REGION Network 2: Выключение и обнуление таймера
   RUNG wire#powerrail
      I_Contact( #Start )
      wire#w1
      { S7_GenerateENO := "TRUE" } Move(in := 0, out1 => #Now)
      wire#w2
      R_Coil( #"Exit" )
   END_RUNG
   RUNG wire#powerrail
      Contact( #Reset )
   END_RUNG wire#w1
   RUNG wire#powerrail
      { S7_Templates := "SrcType := Int" } LT_Contact(in1 := #Now, in2 := #SP)
   END_RUNG wire#w2
   RUNG wire#w2
      R_Coil( #Reset )
   END_RUNG
   // the same network as SCL:
   // ENO of a box is taken as its EN; it also drops when the box reports an error
   #_w1 := NOT #Start OR #Reset;
   IF #_w1 THEN #Now := 0; END_IF;
   IF #_w1 OR (#Now < #SP) THEN
       #"Exit" := FALSE;
       #Reset := FALSE;
   END_IF;
END_REGION
END_FUNCTION_BLOCK

FUNCTION "Modbus_KP" : Void
{ S7_Optimized_Access := 'TRUE' }
VERSION : 0.1
   VAR_INPUT 
      KP : Int;
      cnt : Int;
   END_VAR

   VAR_OUTPUT 
      use : Bool;
   END_VAR

   VAR_IN_OUT 
      IP {InstructionName := 'IP_V4'; LibVersion := '1.0'} : IP_V4;
      Port : UInt;
      ADDR : UInt;
   END_VAR


BEGIN
	CASE #KP OF
	    1:  //  КП2.1
	        IF NOT "AUMA_KP_2_1_DB".AUMA[#cnt].Use THEN
	            "AUMA_KP_2_1_DB".AUMA[#cnt].Link := FALSE;
	            #use := FALSE;
	        ELSE
	            #use := TRUE;
	            #IP := "tGw_DB".tGw["AUMA_KP_2_1_DB".AUMA[#cnt].ID].IP;
	            #Port := "tGw_DB".tGw["AUMA_KP_2_1_DB".AUMA[#cnt].ID]."Port";
	            #ADDR := "AUMA_KP_2_1_DB".AUMA[#cnt].ADDR;
	        END_IF;
	    2:  //  КП2.2
	        IF NOT "AUMA_KP_2_2_DB".AUMA[#cnt].Use THEN
	            "AUMA_KP_2_2_DB".AUMA[#cnt].Link := FALSE;
	            #use := FALSE;
	        ELSE
	            #use := TRUE;
	            #IP := "tGw_DB".tGw["AUMA_KP_2_2_DB".AUMA[#cnt].ID].IP;
	            #Port := "tGw_DB".tGw["AUMA_KP_2_2_DB".AUMA[#cnt].ID]."Port";
	            #ADDR := "AUMA_KP_2_2_DB".AUMA[#cnt].ADDR;
	        END_IF;
	    3:  //  КП2.3
	        IF NOT "AUMA_KP_2_3_DB".AUMA[#cnt].Use THEN
	            "AUMA_KP_2_3_DB".AUMA[#cnt].Link := FALSE;
	            #use := FALSE;
	        ELSE
	            #use := TRUE;
	            #IP := "tGw_DB".tGw["AUMA_KP_2_3_DB".AUMA[#cnt].ID].IP;
	            #Port := "tGw_DB".tGw["AUMA_KP_2_3_DB".AUMA[#cnt].ID]."Port";
	            #ADDR := "AUMA_KP_2_3_DB".AUMA[#cnt].ADDR;
	        END_IF;
	    4:  //  КП2.4
	        IF NOT "AUMA_KP_2_4_DB".AUMA[#cnt].Use THEN
	            "AUMA_KP_2_4_DB".AUMA[#cnt].Link := FALSE;
	            #use := FALSE;
	        ELSE
	            #use := TRUE;
	            #IP := "tGw_DB".tGw["AUMA_KP_2_4_DB".AUMA[#cnt].ID].IP;
	            #Port := "tGw_DB".tGw["AUMA_KP_2_4_DB".AUMA[#cnt].ID]."Port";
	            #ADDR := "AUMA_KP_2_4_DB".AUMA[#cnt].ADDR;
	        END_IF;
	    5:  //  КП2.5
	        IF NOT "AUMA_KP_2_5_DB".AUMA[#cnt].Use THEN
	            "AUMA_KP_2_5_DB".AUMA[#cnt].Link := FALSE;
	            #use := FALSE;
	        ELSE
	            #use := TRUE;
	            #IP := "tGw_DB".tGw["AUMA_KP_2_5_DB".AUMA[#cnt].ID].IP;
	            #Port := "tGw_DB".tGw["AUMA_KP_2_5_DB".AUMA[#cnt].ID]."Port";
	            #ADDR := "AUMA_KP_2_5_DB".AUMA[#cnt].ADDR;
	        END_IF;
	    6:  //  КП2.6
	        IF NOT "AUMA_KP_2_6_DB".AUMA[#cnt].Use THEN
	            "AUMA_KP_2_6_DB".AUMA[#cnt].Link := FALSE;
	            #use := FALSE;
	        ELSE
	            #use := TRUE;
	            #IP := "tGw_DB".tGw["AUMA_KP_2_6_DB".AUMA[#cnt].ID].IP;
	            #Port := "tGw_DB".tGw["AUMA_KP_2_6_DB".AUMA[#cnt].ID]."Port";
	            #ADDR := "AUMA_KP_2_6_DB".AUMA[#cnt].ADDR;
	        END_IF;
	    7:  //  КП2.7
	        IF NOT "AUMA_KP_2_7_DB".AUMA[#cnt].Use THEN
	            "AUMA_KP_2_7_DB".AUMA[#cnt].Link := FALSE;
	            #use := FALSE;
	        ELSE
	            #use := TRUE;
	            #IP := "tGw_DB".tGw["AUMA_KP_2_7_DB".AUMA[#cnt].ID].IP;
	            #Port := "tGw_DB".tGw["AUMA_KP_2_7_DB".AUMA[#cnt].ID]."Port";
	            #ADDR := "AUMA_KP_2_7_DB".AUMA[#cnt].ADDR;
	        END_IF;
	    8:  //  КП2.8
	        IF NOT "AUMA_KP_2_8_DB".AUMA[#cnt].Use THEN
	            "AUMA_KP_2_8_DB".AUMA[#cnt].Link := FALSE;
	            #use := FALSE;
	        ELSE
	            #use := TRUE;
	            #IP := "tGw_DB".tGw["AUMA_KP_2_8_DB".AUMA[#cnt].ID].IP;
	            #Port := "tGw_DB".tGw["AUMA_KP_2_8_DB".AUMA[#cnt].ID]."Port";
	            #ADDR := "AUMA_KP_2_8_DB".AUMA[#cnt].ADDR;
	        END_IF;
	    9:  //  КП2.9
	        IF NOT "AUMA_KP_2_9_DB".AUMA[#cnt].Use THEN
	            "AUMA_KP_2_9_DB".AUMA[#cnt].Link := FALSE;
	            #use := FALSE;
	        ELSE
	            #use := TRUE;
	            #IP := "tGw_DB".tGw["AUMA_KP_2_9_DB".AUMA[#cnt].ID].IP;
	            #Port := "tGw_DB".tGw["AUMA_KP_2_9_DB".AUMA[#cnt].ID]."Port";
	            #ADDR := "AUMA_KP_2_9_DB".AUMA[#cnt].ADDR;
	        END_IF;
	    10:  //  КП2.10
	        IF NOT "AUMA_KP_2_10_DB".AUMA[#cnt].Use THEN
	            "AUMA_KP_2_10_DB".AUMA[#cnt].Link := FALSE;
	            #use := FALSE;
	        ELSE
	            #use := TRUE;
	            #IP := "tGw_DB".tGw["AUMA_KP_2_10_DB".AUMA[#cnt].ID].IP;
	            #Port := "tGw_DB".tGw["AUMA_KP_2_10_DB".AUMA[#cnt].ID]."Port";
	            #ADDR := "AUMA_KP_2_10_DB".AUMA[#cnt].ADDR;
	        END_IF;
	    11:  //  КП1
	        IF NOT "AUMA_KP_1_DB".AUMA[#cnt].Use THEN
	            "AUMA_KP_1_DB".AUMA[#cnt].Link := FALSE;
	            #use := FALSE;
	        ELSE
	            #use := TRUE;
	            #IP := "tGw_DB".tGw["AUMA_KP_1_DB".AUMA[#cnt].ID].IP;
	            #Port := "tGw_DB".tGw["AUMA_KP_1_DB".AUMA[#cnt].ID]."Port";
	            #ADDR := "AUMA_KP_1_DB".AUMA[#cnt].ADDR;
	        END_IF;
	    ELSE
	        #use := FALSE;
	END_CASE;
END_FUNCTION

FUNCTION "ModBus_AUMA_READ" : Void
{ S7_Optimized_Access := 'TRUE' }
VERSION : 0.1
   VAR_TEMP 
      offset : UInt;
      "DB" : UInt;
   END_VAR


BEGIN
	IF "ModBus_DB".cnt > 0 THEN
	    #offset := ("ModBus_DB".cnt * 40);
	ELSE
	    #offset := 0;
	END_IF;
	
	#DB := 410 + "ModBus_DB".KP;
	
	CASE "ModBus_DB".KP OF
	    1:
	        "AUMA_KP_2_1_DB".AUMA["ModBus_DB".cnt].Link := TRUE;
	        "ModBus_DB".update := "AUMA_KP_2_1_DB".AUMA["ModBus_DB".cnt].Update;
	    2:
	        "AUMA_KP_2_2_DB".AUMA["ModBus_DB".cnt].Link := TRUE;
	        "ModBus_DB".update := "AUMA_KP_2_2_DB".AUMA["ModBus_DB".cnt].Update;
	    3:
	        "AUMA_KP_2_3_DB".AUMA["ModBus_DB".cnt].Link := TRUE;
	        "ModBus_DB".update := "AUMA_KP_2_3_DB".AUMA["ModBus_DB".cnt].Update;
	    4:
	        "AUMA_KP_2_4_DB".AUMA["ModBus_DB".cnt].Link := TRUE;
	        "ModBus_DB".update := "AUMA_KP_2_4_DB".AUMA["ModBus_DB".cnt].Update;
	    5:
	        "AUMA_KP_2_5_DB".AUMA["ModBus_DB".cnt].Link := TRUE;
	        "ModBus_DB".update := "AUMA_KP_2_5_DB".AUMA["ModBus_DB".cnt].Update;
	    6:
	        "AUMA_KP_2_6_DB".AUMA["ModBus_DB".cnt].Link := TRUE;
	        "ModBus_DB".update := "AUMA_KP_2_6_DB".AUMA["ModBus_DB".cnt].Update;
	    7:
	        "AUMA_KP_2_7_DB".AUMA["ModBus_DB".cnt].Link := TRUE;
	        "ModBus_DB".update := "AUMA_KP_2_7_DB".AUMA["ModBus_DB".cnt].Update;
	    8:
	        "AUMA_KP_2_8_DB".AUMA["ModBus_DB".cnt].Link := TRUE;
	        "ModBus_DB".update := "AUMA_KP_2_8_DB".AUMA["ModBus_DB".cnt].Update;
	    9:
	        "AUMA_KP_2_9_DB".AUMA["ModBus_DB".cnt].Link := TRUE;
	        "ModBus_DB".update := "AUMA_KP_2_9_DB".AUMA["ModBus_DB".cnt].Update;
	    10:
	        "AUMA_KP_2_10_DB".AUMA["ModBus_DB".cnt].Link := TRUE;
	        "ModBus_DB".update := "AUMA_KP_2_10_DB".AUMA["ModBus_DB".cnt].Update;
	    11:
	        "AUMA_KP_1_DB".AUMA["ModBus_DB".cnt].Link := TRUE;
	        "ModBus_DB".update := "AUMA_KP_1_DB".AUMA["ModBus_DB".cnt].Update;
	    12:
	        "AUMA_KP_2_DB".AUMA["ModBus_DB".cnt].Link := TRUE;
	        "ModBus_DB".update := "AUMA_KP_2_DB".AUMA["ModBus_DB".cnt].Update;
	    13:
	        "AUMA_KP_3_DB".AUMA["ModBus_DB".cnt].Link := TRUE;
	        "ModBus_DB".update := "AUMA_KP_3_DB".AUMA["ModBus_DB".cnt].Update;
	    14:
	        "AUMA_KP_4_DB".AUMA["ModBus_DB".cnt].Link := TRUE;
	        "ModBus_DB".update := "AUMA_KP_4_DB".AUMA["ModBus_DB".cnt].Update;
	    15:
	        "AUMA_KP_5_DB".AUMA["ModBus_DB".cnt].Link := TRUE;
	        "ModBus_DB".update := "AUMA_KP_5_DB".AUMA["ModBus_DB".cnt].Update;
	END_CASE;
	
	"Indirect_MOVE"(
	                Length := 4,
	                Source_DB := 40,
	                Source_OFFSET := 0,
	                Target_DB := #DB,
	                Target_OFFSET := #offset);
END_FUNCTION

FUNCTION "ModBus_AUMA_ERROR" : Void
{ S7_Optimized_Access := 'TRUE' }
VERSION : 0.1
   VAR_TEMP 
      offset : UInt;
      "DB" : UInt;
   END_VAR


BEGIN
	CASE "ModBus_DB".KP OF
	    1:
	        "AUMA_KP_2_1_DB".AUMA["ModBus_DB".cnt].Link := FALSE;
	        "AUMA_KP_2_1_DB".AUMA["ModBus_DB".cnt].NoRead := TRUE;
	    2:
	        "AUMA_KP_2_2_DB".AUMA["ModBus_DB".cnt].Link := FALSE;
	        "AUMA_KP_2_2_DB".AUMA["ModBus_DB".cnt].NoRead := TRUE;
	    3:
	        "AUMA_KP_2_3_DB".AUMA["ModBus_DB".cnt].Link := FALSE;
	        "AUMA_KP_2_3_DB".AUMA["ModBus_DB".cnt].NoRead := TRUE;
	    4:
	        "AUMA_KP_2_4_DB".AUMA["ModBus_DB".cnt].Link := FALSE;
	        "AUMA_KP_2_4_DB".AUMA["ModBus_DB".cnt].NoRead := TRUE;
	    5:
	        "AUMA_KP_2_5_DB".AUMA["ModBus_DB".cnt].Link := FALSE;
	        "AUMA_KP_2_5_DB".AUMA["ModBus_DB".cnt].NoRead := TRUE;
	    6:
	        "AUMA_KP_2_6_DB".AUMA["ModBus_DB".cnt].Link := FALSE;
	        "AUMA_KP_2_6_DB".AUMA["ModBus_DB".cnt].NoRead := TRUE;
	    7:
	        "AUMA_KP_2_7_DB".AUMA["ModBus_DB".cnt].Link := FALSE;
	        "AUMA_KP_2_7_DB".AUMA["ModBus_DB".cnt].NoRead := TRUE;
	    8:
	        "AUMA_KP_2_8_DB".AUMA["ModBus_DB".cnt].Link := FALSE;
	        "AUMA_KP_2_8_DB".AUMA["ModBus_DB".cnt].NoRead := TRUE;
	    9:
	        "AUMA_KP_2_9_DB".AUMA["ModBus_DB".cnt].Link := FALSE;
	        "AUMA_KP_2_9_DB".AUMA["ModBus_DB".cnt].NoRead := TRUE;
	    10:
	        "AUMA_KP_2_10_DB".AUMA["ModBus_DB".cnt].Link := FALSE;
	        "AUMA_KP_2_10_DB".AUMA["ModBus_DB".cnt].NoRead := TRUE;
	    11:
	        "AUMA_KP_1_DB".AUMA["ModBus_DB".cnt].Link := FALSE;
	        "AUMA_KP_1_DB".AUMA["ModBus_DB".cnt].NoRead := TRUE;
	    12:
	        "AUMA_KP_2_DB".AUMA["ModBus_DB".cnt].Link := FALSE;
	        "AUMA_KP_2_DB".AUMA["ModBus_DB".cnt].NoRead := TRUE;
	    13:
	        "AUMA_KP_3_DB".AUMA["ModBus_DB".cnt].Link := FALSE;
	        "AUMA_KP_3_DB".AUMA["ModBus_DB".cnt].NoRead := TRUE;
	    14:
	        "AUMA_KP_4_DB".AUMA["ModBus_DB".cnt].Link := FALSE;
	        "AUMA_KP_4_DB".AUMA["ModBus_DB".cnt].NoRead := TRUE;
	    15:
	        "AUMA_KP_5_DB".AUMA["ModBus_DB".cnt].Link := FALSE;
	        "AUMA_KP_5_DB".AUMA["ModBus_DB".cnt].NoRead := TRUE;
	    20:
	        "FE_DB".FE["ModBus_DB".cnt].Link := FALSE;
	        "FE_DB".FE["ModBus_DB".cnt].NoRead := TRUE;
	    21:
	        "LE_DB".LE["ModBus_DB".cnt].Link := FALSE;
	        "LE_DB".LE["ModBus_DB".cnt].NoRead := TRUE;
	    22:
	        "PE_DB".PE["ModBus_DB".cnt].Link := FALSE;
	        "PE_DB".PE["ModBus_DB".cnt].NoRead := TRUE;
	END_CASE;
	
	
END_FUNCTION

FUNCTION "ModBus_AUMA_WRITE" : Void
{ S7_Optimized_Access := 'TRUE' }
VERSION : 0.1
   VAR_TEMP 
      offset : UInt;
      "DB" : UInt;
   END_VAR

   VAR CONSTANT 
      I : Byte := 16#81;   // Input
      Q : Byte := 16#82;   // Output
      M : Byte := 16#83;   // Bit Memory
      D : Byte := 16#84;   // Data Block
      PIW : Byte := 16#1;   // S7-1500 Only
      zero : Byte;
   END_VAR


BEGIN
	IF "ModBus_DB".cnt > 0 THEN
	    #offset := ("ModBus_DB".cnt * 40);
	ELSE
	    #offset := 0;
	END_IF;
	
	#DB := 410 + "ModBus_DB".KP;
	
	//запись команды и уставки в коммуникацию
	"Indirect_MOVE"(
	                Length := 2,
	                Source_DB := #DB,
	                Source_OFFSET := #offset + 14,
	                Target_DB := 40,
	                Target_OFFSET := 0);
END_FUNCTION

FUNCTION_BLOCK "ModBus_TCP"   // FB40, LAD
TITLE = Блок опроса ModBus TCP
{ S7_Optimized_Access := 'FALSE' }
VERSION : 0.1
// ВНИМАНИЕ!  Через один аппаратный порт контроллера можно проводить множество различных опросов по ModBus TCP. Для этого у каждого экземпляра должен быть указан уникальный CONNECT.ID.
// 
// Для каждого уникального CONNECT.ID / внешней ветки / точки подключения (IP, RemotePort) рекомендуется использовать отдельный экземпляр функционального блока. Например, при использовании tGW-735 имеющего 3 порта подключения с RemotePort = 502, 503 и 504 соответственно (но общий IP адрес) рекомендуется использовать три отдельных блока ModBus_TCP с уникальными CONNECT.ID.
// 
// Каждая точка чтения/записи = 1 экземпляр DEV_Config, количество элементов в массиве можно менять по необходимости, итоговое количество элементов массива указывается в теге Limit.
// 
// Для режима чтения необходимо указать:
// - MODE = 0
// - Source_DB = 40 (номер DB Modbus_TCP_DB)
// - SourceOFFSET = 0
// - Target_DB = xx (номер DB, куда необходимо положить прочитанные данные)
// - Target_OFFSET = xx (номер байта, начиная с которого кладутся прочитанные данные в выбранный DB)
// 
// Для режима опроса необходимо указать:
// - MODE = 1
// - Source_DB = xx (номер DB, откуда необходимо взять данные для передачи)
// - Source_OFFSET = xx (номер байта, начиная с которого берутся данные для передачи)
// - Target_DB = 40 (номер DB Modbus_TCP_DB)
// - Target_OFFSET = 0
// stored: AutoNumber false, IsIECCheckEnabled false, SetENOAutomatically false, UDAEnableTagReadback false
   VAR DB_SPECIFIC
      DATA : Array[0..100] of Word;   // Массив данных
      CONNECT { S7_SetPoint := 'True'} : TCON_IP_v4;
   END_VAR
   // CONNECT.InterfaceId := 64;
   // CONNECT.ID := 16#0001;
   // CONNECT.ConnectionType := 16#0B;
   // CONNECT.ActiveEstablished := TRUE;
   // CONNECT.RemoteAddress.ADDR[1] := 16#C0;
   // CONNECT.RemoteAddress.ADDR[2] := 16#A8;
   // CONNECT.RemoteAddress.ADDR[3] := 16#00;
   // CONNECT.RemoteAddress.ADDR[4] := 16#0A;
   // CONNECT.RemotePort := 502;
   // CONNECT.LocalPort := 0;
BEGIN

REGION Network 1
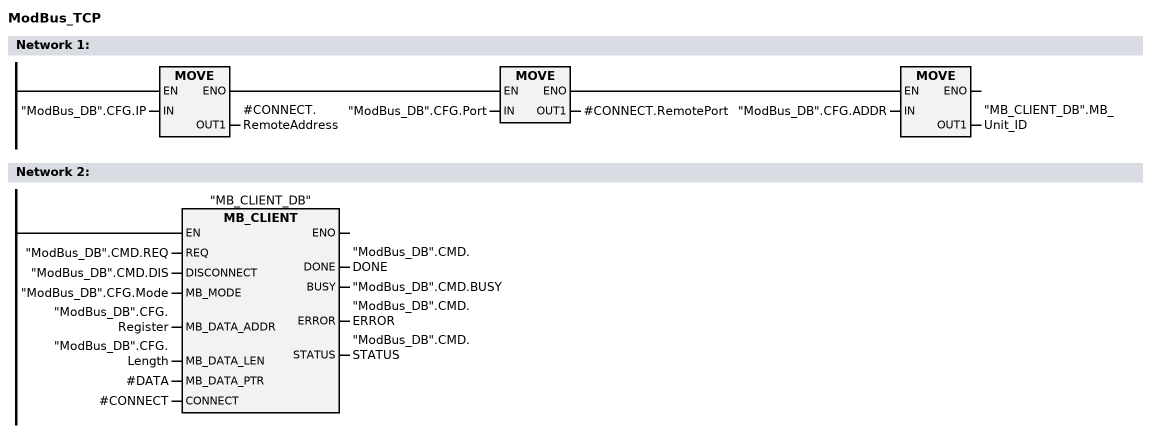
   RUNG wire#powerrail
      Move(in := "ModBus_DB".CFG.IP, out1 => #CONNECT.RemoteAddress)
      Move(in := "ModBus_DB".CFG.Port, out1 => #CONNECT.RemotePort)
      Move(in := "ModBus_DB".CFG.ADDR, out1 => "MB_CLIENT_DB".MB_Unit_ID)
   END_RUNG
   // the same network as SCL:
   #CONNECT.RemoteAddress := "ModBus_DB".CFG.IP;
   #CONNECT.RemotePort := "ModBus_DB".CFG.Port;
   "MB_CLIENT_DB".MB_Unit_ID := "ModBus_DB".CFG.ADDR;
END_REGION

REGION Network 2
   RUNG wire#powerrail
      "MB_CLIENT_DB".MB_CLIENT(REQ := "ModBus_DB".CMD.REQ, DISCONNECT := "ModBus_DB".CMD.DIS, MB_MODE := "ModBus_DB".CFG.Mode, MB_DATA_ADDR := "ModBus_DB".CFG.Register, MB_DATA_LEN := "ModBus_DB".CFG.Length, MB_DATA_PTR := #DATA, CONNECT := #CONNECT, DONE => "ModBus_DB".CMD.DONE, BUSY => "ModBus_DB".CMD.BUSY, ERROR => "ModBus_DB".CMD.ERROR, STATUS => "ModBus_DB".CMD.STATUS)
   END_RUNG
   // the same network as SCL:
   "MB_CLIENT_DB"(REQ := "ModBus_DB".CMD.REQ,   // MB_CLIENT
                  DISCONNECT := "ModBus_DB".CMD.DIS,
                  MB_MODE := "ModBus_DB".CFG.Mode,
                  MB_DATA_ADDR := "ModBus_DB".CFG.Register,
                  MB_DATA_LEN := "ModBus_DB".CFG.Length,
                  MB_DATA_PTR := #DATA,
                  CONNECT := #CONNECT,
                  DONE => "ModBus_DB".CMD.DONE,
                  BUSY => "ModBus_DB".CMD.BUSY,
                  ERROR => "ModBus_DB".CMD.ERROR,
                  STATUS => "ModBus_DB".CMD.STATUS);
END_REGION
END_FUNCTION_BLOCK

FUNCTION_BLOCK "SKV_Main"
{ S7_Optimized_Access := 'FALSE' }
VERSION : 0.1
   VAR 
      One : Array[0..11] of "SKV_One";
      SP : Struct   // Уставки
         Max { S7_SetPoint := 'True'} : Real;   // - максимальная производительность
         High : Real;   // - высокая производительность
         Auto : Real;   // - рабочая уставка
         Point : Real;   // - сниженная производительность
         Low : Real;   // - низкая производительность
         Min { S7_SetPoint := 'True'} : Real;   // - минимальная производительность
      END_STRUCT;
      cnt : Struct   // счетчики
         Min { S7_SetPoint := 'True'} : Int;   // - минимальное кол-во устр-в
         Fix { S7_SetPoint := 'True'} : Int := 2;   // - кол-во устр-в в фиксированном режиме
         All : Int;   // - кол-во устройств общее
         Group : Int;   // - кол-во основных устройств
         Reserve : Int;   // - кол-во резервных устройств
         Ready : Int;   // - кол-во готовых устройств
         Low : Int;   // - кол-во устр-в на сниженной скорости
         Work : Int;   // - кол-во запущенных устройств
         Start : Int;   // - кол-во устр-в в работе
      END_STRUCT;
      tmp : Int;
   END_VAR


BEGIN
	//Распредление нагрузки
	"SKV_Load"(Add_REQ :="SKV_cnt_DB".CMD.Add,
	           Add_Ready => "SKV_cnt_DB".Data.Add_Ready,
	           cnt := #tmp);
	
	//Управление запуском и остановом
	"SKV_cnt_DB"();
	
	//Выбор кол-ва устр-в
	"SKV_Logic_DB"();
	
	//Проверка готовности маршрутов
	"Route_Check_DB"();
	
	//управление маршрутами
	"Route_Control_DB"();
	
	REGION "SKV_One"
	    // Вызов управления каждой скважиной
	    #One[1](Ready:= "Comm_SKV_1".From_SKV.STATE.Ready,
	            Warning:= "Comm_SKV_1".From_SKV.STATE.Warning,
	            Alarm:= "Comm_SKV_1".From_SKV.STATE.Alarm,
	            Route:="Comm_SKV_1".Route,
	            FeedBack := "Comm_SKV_1".FE,
	            REQ_CMD=> "Comm_SKV_1".To_SKV.CMD.REQ,
	            REQ_SP=> "Comm_SKV_1".SP_FE);
	    #One[2](Ready := "Comm_SKV_2".From_SKV.STATE.Ready,
	            Warning := "Comm_SKV_2".From_SKV.STATE.Warning,
	            Alarm := "Comm_SKV_2".From_SKV.STATE.Alarm,
	            Route := "Comm_SKV_2".Route,
	            FeedBack := "Comm_SKV_2".FE,
	            REQ_CMD => "Comm_SKV_2".To_SKV.CMD.REQ,
	            REQ_SP => "Comm_SKV_2".SP_FE);
	    #One[3](Ready := "Comm_SKV_3".From_SKV.STATE.Ready,
	            Warning := "Comm_SKV_3".From_SKV.STATE.Warning,
	            Alarm := "Comm_SKV_3".From_SKV.STATE.Alarm,
	            Route := "Comm_SKV_3".Route,
	            FeedBack := "Comm_SKV_3".FE,
	            REQ_CMD => "Comm_SKV_3".To_SKV.CMD.REQ,
	            REQ_SP => "Comm_SKV_3".SP_FE);
	    #One[4](Ready := "Comm_SKV_12".From_SKV.STATE.Ready,
	            Warning := "Comm_SKV_12".From_SKV.STATE.Warning,
	            Alarm := "Comm_SKV_12".From_SKV.STATE.Alarm,
	            Route := "Comm_SKV_12".Route,
	            FeedBack := "Comm_SKV_12".FE,
	            REQ_CMD => "Comm_SKV_12".To_SKV.CMD.REQ,
	            REQ_SP => "Comm_SKV_12".SP_FE);
	    #One[5](Ready := "Comm_SKV_13".From_SKV.STATE.Ready,
	            Warning := "Comm_SKV_13".From_SKV.STATE.Warning,
	            Alarm := "Comm_SKV_13".From_SKV.STATE.Alarm,
	            Route := "Comm_SKV_13".Route,
	            FeedBack := "Comm_SKV_13".FE,
	            REQ_CMD => "Comm_SKV_13".To_SKV.CMD.REQ,
	            REQ_SP => "Comm_SKV_13".SP_FE);
	    #One[6](Ready := "Comm_SKV_14".From_SKV.STATE.Ready,
	            Warning := "Comm_SKV_14".From_SKV.STATE.Warning,
	            Alarm := "Comm_SKV_14".From_SKV.STATE.Alarm,
	            Route := "Comm_SKV_14".Route,
	            FeedBack := "Comm_SKV_14".FE,
	            REQ_CMD => "Comm_SKV_14".To_SKV.CMD.REQ,
	            REQ_SP => "Comm_SKV_14".SP_FE);
	    #One[7](Ready := "Comm_SKV_15".From_SKV.STATE.Ready,
	            Warning := "Comm_SKV_15".From_SKV.STATE.Warning,
	            Alarm := "Comm_SKV_15".From_SKV.STATE.Alarm,
	            Route := "Comm_SKV_15".Route,
	            FeedBack := "Comm_SKV_15".FE,
	            REQ_CMD => "Comm_SKV_15".To_SKV.CMD.REQ,
	            REQ_SP => "Comm_SKV_15".SP_FE);
	    #One[8](Ready := "Comm_SKV_20".From_SKV.STATE.Ready,
	            Warning := "Comm_SKV_20".From_SKV.STATE.Warning,
	            Alarm := "Comm_SKV_20".From_SKV.STATE.Alarm,
	            Route := "Comm_SKV_20".Route,
	            FeedBack := "Comm_SKV_20".FE,
	            REQ_CMD => "Comm_SKV_20".To_SKV.CMD.REQ,
	            REQ_SP => "Comm_SKV_20".SP_FE);
	    #One[9](Ready := "Comm_SKV_21".From_SKV.STATE.Ready,
	            Warning := "Comm_SKV_21".From_SKV.STATE.Warning,
	            Alarm := "Comm_SKV_21".From_SKV.STATE.Alarm,
	            Route := "Comm_SKV_21".Route,
	            FeedBack := "Comm_SKV_21".FE,
	            REQ_CMD => "Comm_SKV_21".To_SKV.CMD.REQ,
	            REQ_SP => "Comm_SKV_21".SP_FE);
	    #One[10](Ready := "Comm_SKV_22".From_SKV.STATE.Ready,
	             Warning := "Comm_SKV_22".From_SKV.STATE.Warning,
	             Alarm := "Comm_SKV_22".From_SKV.STATE.Alarm,
	             Route := "Comm_SKV_22".Route,
	             FeedBack := "Comm_SKV_22".FE,
	             REQ_CMD => "Comm_SKV_22".To_SKV.CMD.REQ,
	             REQ_SP => "Comm_SKV_22".SP_FE);
	    #One[11](Ready := "Comm_SKV_23".From_SKV.STATE.Ready,
	             Warning := "Comm_SKV_23".From_SKV.STATE.Warning,
	             Alarm := "Comm_SKV_23".From_SKV.STATE.Alarm,
	             Route := "Comm_SKV_23".Route,
	             FeedBack := "Comm_SKV_23".FE,
	             REQ_CMD => "Comm_SKV_23".To_SKV.CMD.REQ,
	             REQ_SP => "Comm_SKV_23".SP_FE);
	END_REGION
	
END_FUNCTION_BLOCK

FUNCTION_BLOCK "SKV_One"
{ S7_Optimized_Access := 'FALSE' }
VERSION : 0.1
   VAR_INPUT 
      Ready : Bool;   // Флаг готовности устр-ва
      Warning : Bool;   // Флаг предупрждения
      Alarm : Bool;   // Флаг аварии устр-ва
      Route : Bool;   // Флаг готовности маршрута
      FeedBack : Real;   // ОС производительности утр-ва
   END_VAR

   VAR_OUTPUT 
      REQ_CMD : Bool;   // Команда - запуск устр-ва
      REQ_SP : Real;   // Команда - уставка производительности устр-ва
   END_VAR

   VAR 
      Enable : Bool;   // Флаг выбора устр-ва для работы
      SP_Use { S7_SetPoint := 'True'} : Bool := true;   // Использовать флаг достижения уставки
      CMD { S7_SetPoint := 'False'} : "CMD";   // Управляющее слово
      Mode { S7_SetPoint := 'True'} : Int;   // Режим работы
      Status : Int;   // Статус устр-ва
      C { S7_SetPoint := 'True'} : Real;   // Коэффециент эффективности
      Delta : Real;   // Текущее отклонение от уставки
      SP : Struct   // Уставки
         Ok : Bool;   // Флаг достижения уставки
         Auto : Real;   // - авто режим
         Hand : Real;   // - ручной режим
         Low_Percent { S7_SetPoint := 'True'} : Real := 85.0;   // - замедление до %
         Low : Real;   // - замедленная скорость
         Min { S7_SetPoint := 'True'} : Real := 30.0;   // - минимальный расход
         Max { S7_SetPoint := 'True'} : Real := 45.0;   // - максимальный расход
         Delta { S7_SetPoint := 'True'} : Real := 10.0;   // - допустимое отклонение
         Last : Real;   // - прошлая уставка
      END_STRUCT;
      drv_CMD { S7_SetPoint := 'False'} : "drv_CMD";
      support : Word;
      PT {InstructionName := 'R_TRIG'; LibVersion := '1.0'; S7_SetPoint := 'False'} : Array[0..1] of R_TRIG;
      NT {InstructionName := 'F_TRIG'; LibVersion := '1.0'; S7_SetPoint := 'False'} : Array[0..1] of F_TRIG;
   END_VAR


BEGIN
	//Управление одной скважиной
	
	#CMD.Lock := NOT #Ready OR #Alarm;  //Запрет запуска
	#CMD.Ready := NOT #CMD.Lock;
	
	//Ограничение уставки
	IF NOT #CMD.Hand THEN
	    #SP.Hand := #SP.Auto;
	END_IF;
	IF #SP.Hand < #SP.Min THEN
	    #SP.Hand := #SP.Min;
	END_IF;
	IF #SP.Hand > #SP.Max THEN
	    #SP.Hand := #SP.Max;
	END_IF;
	
	//Замедленная скорость
	#SP.Low := #SP.Hand * (100 / #SP.Low_Percent);
	
	//Контроль достижения уставки
	IF #SP.Last <> #SP.Hand THEN
	    #Delta := ABS(#SP.Hand - #SP.Last);
	    IF #Delta < #SP.Delta THEN
	        #SP.Last := #SP.Hand;
	        #SP.Ok := TRUE;
	    ELSE
	        #SP.Ok := FALSE;
	    END_IF;
	END_IF;
	#PT[0](CLK := #SP.Ok);
	
	//device control
	#drv_CMD(Emergency := #support.%X0,
	          CMD := #CMD);
	 //manual mode flag
	     IF #CMD.Hand THEN
	         "Hand_MDA" := TRUE;
	     END_IF;
	     
	//Отключение
	     IF NOT #CMD.Start_M AND #Mode > 1 AND #Mode <= 5 THEN
	         IF #Status <> 5 THEN
	             #Mode := 5;
	         ELSE
	             #Mode := 6;
	         END_IF;
	     END_IF;
	     
	//Режимы работы
	     CASE #Mode OF
	         0: //Установка отключена
	             #CMD.Start_A := FALSE;
	             #CMD.Start_M := FALSE;
	             #Status := 0;
	             #Mode := 1;
	         1: //Запуск в работу
	             IF #CMD.Start_M THEN
	                 #REQ_CMD := TRUE;
	                 #REQ_SP := #SP.Min;
	                 IF #Status = 0 THEN
	                     #Status := 10; //выход на минимальную рабочую точку
	                 ELSIF #Status = 10 AND (#PT[0].Q OR NOT #SP_Use) THEN
	                     #Status := 1;  //готов к работе
	                 END_IF;
	             ELSE
	                 #REQ_CMD := FALSE;
	                 #REQ_SP := 0.0;
	                 #Status := 0;
	             END_IF;
	         2:  //Плавный разгон до общей точки
	             IF #Status = 1 THEN
	                 #REQ_SP := #SP.Hand;
	                 #Status := 20;     //выход на общую рабочую точку
	             ELSIF #Status = 20 AND (#PT[0].Q OR NOT #SP_Use) THEN
	                 #Status := 2;      //рабочая точка достигнута
	             END_IF;
	         3:  //Переход в штатный режим работы
	             IF #Status = 2 OR #Status = 4 THEN
	                 #Status := 3;       //штатный режим работы
	             ELSIF #Status = 3 THEN
	                 IF NOT #Warning THEN
	                     #REQ_SP := #SP.Hand;
	                 ELSE
	                     #REQ_SP := #SP.Low;
	                 END_IF;
	             END_IF;
	         4: //Замедление перед вводном нового элемента в работу
	             IF #Status = 3 THEN
	                 #REQ_SP := #SP.Hand;
	                 #Status := 40;        //замедление при вводе нового элемента
	             ELSIF #Status = 40 AND (#PT[0].Q OR NOT #SP_Use) THEN
	                 #Status := 4;
	             END_IF;
	         5: //Замедление при отключении
	             IF #Status <> 50 AND #Status <> 5 THEN
	                 #REQ_SP := #SP.Min;
	                 #Status := 50;
	             ELSIF #Status = 50 AND (NOT #Enable OR #CMD.Lock OR (#PT[0].Q OR NOT #SP_Use)) THEN
	                 #Status := 5;
	             END_IF;
	         6: //Вывод элемента из работы
	             IF #Status = 5 THEN
	                 #CMD.Start_A := FALSE;
	                 #REQ_CMD := FALSE;
	                 #REQ_SP := 0.0;
	                 #Status := 60;
	             ELSIF #Status = 60 AND (#PT[0].Q OR NOT #SP_Use) THEN
	                 #Status := 0;
	                 #Mode := 0;
	             END_IF;
	     END_CASE;
	     
	
END_FUNCTION_BLOCK

FUNCTION_BLOCK "drv_CMD"
{ S7_Optimized_Access := 'TRUE' }
VERSION : 0.1
   VAR_INPUT 
      Emergency : Bool;
   END_VAR

   VAR_IN_OUT 
      CMD : "CMD";
   END_VAR


BEGIN
	// Device mode determination
	IF NOT #Emergency THEN
	    //Normal mode
	    IF NOT #CMD.Force THEN
	        //No technological lock
	        IF NOT #CMD.Lock AND NOT #CMD.Alarm THEN
	            //No manual mode
	            IF NOT #CMD.Hand THEN
	                #CMD.Start_M := #CMD.Start_A;
	            END_IF;
	        ELSE
	            //Technological lock or device alarm
	            #CMD.Start_M := FALSE;
	        END_IF;
	    ELSE
	        IF #CMD.Lock OR #CMD.Alarm THEN
	            #CMD.Start_M := FALSE;
	        END_IF;
	    END_IF;
	ELSE
	    //Emergency stop
	    #CMD.Start_M := FALSE;
	END_IF;
END_FUNCTION_BLOCK

FUNCTION "SKV_Load" : Void
{ S7_Optimized_Access := 'TRUE' }
VERSION : 0.1
   VAR_INPUT 
      Add_REQ : Bool;   // Запрос ввода нового устр-ва в работу
   END_VAR

   VAR_OUTPUT 
      Add_Ready : Bool;   // Устр-ва готовы к вводу нового устр-ва в работу
   END_VAR

   VAR_IN_OUT 
      cnt : Int;   // счетчик
   END_VAR

   VAR_TEMP 
      x : Int;
   END_VAR


BEGIN
	//обнуление временных значений
	#Add_Ready := FALSE;
	"SKV_Main_DB".cnt.Ready := 0;
	"SKV_Main_DB".cnt.Low := 0;
	"SKV_Main_DB".cnt.Start := 0;
	"SKV_Main_DB".cnt.Work := 0;
	
	IF "SKV_Main_DB".SP.Auto > "SKV_Main_DB".SP.Max THEN
	    "SKV_Main_DB".SP.Auto := "SKV_Main_DB".SP.Max;
	END_IF;
	
	//вычисление точки схождения скоростей
	"SKV_Main_DB".SP.Point := "SKV_Main_DB".SP.Low + ((("SKV_Main_DB".SP.Auto - "SKV_Main_DB".SP.Low) / "SKV_Main_DB".cnt.Min) * 2);
	
	//Распределение уставки по работающим насосам
	FOR #x := 1 TO "SKV_Main_DB".cnt.All DO
	    
	    //число готовых насосов
	    IF "SKV_Main_DB".One[#x].CMD.Ready THEN
	        "SKV_Main_DB".cnt.Ready := "SKV_Main_DB".cnt.Ready + 1;
	    END_IF;
	    
	    //число насосов в работе
	    IF "SKV_Main_DB".One[#x].CMD.Start_M THEN
	        "SKV_Main_DB".cnt.Start := "SKV_Main_DB".cnt.Start + 1;
	    END_IF;
	    
	    //число насосов в штатном режиме
	    IF "SKV_Main_DB".One[#x].Status = 3 THEN
	        "SKV_Main_DB".cnt.Work := "SKV_Main_DB".cnt.Work + 1;
	    END_IF;
	    
	    //запуск установки
	    IF "SKV_cnt_DB".Step > 0 THEN
	        IF "SKV_cnt_DB".Step < 10 THEN
	            IF "SKV_Main_DB".One[#x].Status = 1 THEN
	                "SKV_Main_DB".One[#x].Mode := 2;
	            END_IF;
	            IF "SKV_Main_DB".One[#x].Status = 2 THEN
	                "SKV_Main_DB".One[#x].Mode := 3;
	            END_IF;
	            "SKV_Main_DB".One[#x].SP.Auto := "SKV_Main_DB".SP.Auto;
	        END_IF;
	    END_IF;
	    
	    //уставка в рабочем режиме
	    IF "SKV_Main_DB".One[#x].Status = 3 OR "SKV_Main_DB".One[#x].Status = 30 THEN
	        "SKV_Main_DB".One[#x].SP.Auto := "SKV_Main_DB".SP.Auto;
	    END_IF;
	    
	  //цикл замедления при подключении нового насоса
	    IF #Add_REQ THEN
	        
	        //команда замедлиться для подключения работающих насосов
	        IF "SKV_Main_DB".One[#x].Status = 3 THEN
	            "SKV_Main_DB".One[#x].Mode := 4;
	        END_IF;
	        
	        //коррекция уставки для замедленных насосов
	        IF "SKV_Main_DB".One[#x].Status = 40 THEN
	            "SKV_Main_DB".One[#x].SP.Auto := "SKV_Main_DB".SP.Point;
	        END_IF;
	        
	        //контроль готовности всех насосов
	        IF "SKV_Main_DB".One[#x].Status = 4 THEN
	            "SKV_Main_DB".cnt.Low := "SKV_Main_DB".cnt.Low + 1;
	            IF "SKV_Main_DB".cnt.Low = #cnt THEN
	                #Add_Ready := true;
	            END_IF;
	        END_IF;
	        
	    END_IF;
	    
	    //возвращение в рабочий режим
	    IF NOT #Add_REQ THEN
	        IF "SKV_Main_DB".One[#x].Status = 4 THEN
	            "SKV_Main_DB".One[#x].Mode := 3;
	        END_IF;
	    END_IF;
	    
	END_FOR;
	
END_FUNCTION

FUNCTION_BLOCK "SKV_Logic"
{ S7_Optimized_Access := 'FALSE' }
VERSION : 0.1
   VAR 
      Start : Bool;   // Команда запуска
      Start_Up { S7_SetPoint := 'True'} : Bool;   // Авто-рестарт
      Mode : Bool;   // Режим работы
      Step : Int;   // шаг операции
      LE : Real;   // Текущий усреднённый уровень
      SP : Struct   // Уставки
         Max { S7_SetPoint := 'True'} : Real;   // - макс уровень
         High { S7_SetPoint := 'True'} : Real;   // - высокий уровень
         Mid { S7_SetPoint := 'True'} : Real;   // - средний уровень
         Low { S7_SetPoint := 'True'} : Real;   // - низкий уровень
         Min { S7_SetPoint := 'True'} : Real;   // - минимальный уровень
      END_STRUCT;
   END_VAR


BEGIN
	//Отключение при первом пуске
	IF NOT #Start_Up AND "FirstScan" THEN
	    #Start := FALSE;
	END_IF;
	
	//Отключение
	IF NOT #Start THEN
	    #Step := 0;
	    "SKV_cnt_DB".CMD.REQ := 0;
	END_IF;
	
	//Общее управление
	CASE #Step OF
	    0:  //Запуск системы
	        IF #Start AND #LE < #SP.Max THEN
	            "SKV_cnt_DB".CMD.REQ := "SKV_Main_DB".cnt.Min;  //минимальное количество устр-в в работе
	            #Step := #Step + 1;
	        END_IF;
	    1:  //проверка режима
	        IF #Mode = 0 THEN
	            #Step := 2; //поддержание уровня
	        ELSIF #Mode = 1 THEN
	            #Step := 3; //фиксированная нагрузка
	        END_IF;
	    2:  //Поддержание уровня
	        IF #LE < #SP.High THEN                              //уровень ниже верхней рабочей точки - вошли в рабочий диапазон
	            IF #LE < #SP.Mid THEN                           //уровень упал ниже среднего - требуется +1 устр-во
	                IF "SKV_cnt_DB".CMD.REQ = "SKV_Main_DB".cnt.Work THEN
	                    IF "SKV_Main_DB".cnt.Work < "SKV_Main_DB".cnt.All AND "SKV_cnt_DB".Step = 10 THEN
	                        "SKV_cnt_DB".CMD.REQ := "SKV_cnt_DB".CMD.REQ + 1;
	                    END_IF;
	                END_IF;
	                IF NOT "SKV_cnt_DB".CMD.Reload AND NOT NOT "SKV_cnt_DB".CMD.Load AND NOT "SKV_cnt_DB".CMD.Rotation AND NOT "SKV_cnt_DB".CMD.Deload AND "SKV_cnt_DB".Step = 10 THEN
	                    IF "SKV_cnt_DB".CMD.REQ > "SKV_Main_DB".cnt.Start THEN
	                        "SKV_cnt_DB".CMD.Reload := TRUE;
	                    END_IF;
	                    IF "SKV_cnt_DB".CMD.REQ < "SKV_Main_DB".cnt.Start THEN
	                        "SKV_cnt_DB".CMD.Deload := TRUE;
	                    END_IF;
	                END_IF;
	            END_IF;
	        ELSE
	            IF "SKV_cnt_DB".CMD.REQ = "SKV_Main_DB".cnt.Work AND "SKV_cnt_DB".Step = 10 THEN
	                "SKV_cnt_DB".CMD.REQ := "SKV_cnt_DB".CMD.REQ - 1;
	                (*IF "SKV_cnt_DB".CMD.REQ < "SKV_Main_DB".cnt.Min THEN
	                    "SKV_cnt_DB".CMD.REQ := "SKV_Main_DB".cnt.Min;
	                END_IF;*)
	                IF "SKV_cnt_DB".CMD.REQ < 0 THEN
	                    "SKV_cnt_DB".CMD.REQ := 0;
	                END_IF;
	            END_IF;
	        END_IF;
	        //Смена режима работы
	        IF #Mode <> 0 THEN
	            #Step := 1;
	        END_IF;
	    3:   //Фиксированный режим
	        IF NOT "SKV_cnt_DB".CMD.Reload AND NOT NOT "SKV_cnt_DB".CMD.Load AND NOT "SKV_cnt_DB".CMD.Rotation AND NOT "SKV_cnt_DB".CMD.Deload AND "SKV_cnt_DB".Step = 10 THEN
	            IF "SKV_cnt_DB".CMD.REQ > "SKV_Main_DB".cnt.Start THEN
	                "SKV_cnt_DB".CMD.Reload := TRUE;
	            END_IF;
	            IF "SKV_cnt_DB".CMD.REQ < "SKV_Main_DB".cnt.Start THEN
	                "SKV_cnt_DB".CMD.Deload := TRUE;
	            END_IF;
	        END_IF;
	        //Смена режима работы
	        IF #Mode <> 1 THEN
	            #Step := 1;
	        END_IF;
	END_CASE;
END_FUNCTION_BLOCK

FUNCTION_BLOCK "KP_2_1"
{ S7_Optimized_Access := 'FALSE' }
VERSION : 0.1
   VAR 
      limit { S7_SetPoint := 'True'} : Int := 2;   // число задвижек в камере
      load : Int;   // отображаемые на экране настройки
      load_last : Int;
      KP : Array[0..10] of "DRV_AUMA";
      load_ok { S7_SetPoint := 'True'} : Bool;
   END_VAR

   VAR_TEMP 
      ID : Int;
      cnt : Int;
   END_VAR


BEGIN
	//дистанционный режим управления
	FOR #cnt := 1 TO #limit BY 1 DO
	    IF "Comm_SKV_2".To_SKV.Valves.Local[0] THEN
	        IF #KP[#cnt].CMD.Hand THEN
	            #KP[#cnt].CMD.Start_M := "Comm_SKV_2".From_SKV.Valves.REQ[#cnt];
	        END_IF;
	        IF "Comm_SKV_2".From_SKV.Valves.REQ[0] THEN
	            #KP[#cnt].CMD.Reset := TRUE;
	            #load := 10;
	        END_IF;
	    ELSE
	        "Comm_SKV_2".To_SKV.Valves.Local[#cnt] := #KP[#cnt].CMD.Start_M;
	    END_IF;
	END_FOR;
	
	//экранный буфер
	"Load_KP_2_1"(last := #load_last,
	              load := #load,
	              ok := #load_ok);
	IF "KP_Reset" THEN
	    #load := 10;
	END_IF;
	
	FOR #cnt := 1 TO #limit BY 1 DO
	    #ID := #KP[#cnt].CodeID;
	    #KP[#cnt].CMD.Local := NOT "AUMA_KP_2_1_DB".AUMA[#ID].Message.Sel_Dist;
	    #KP[#cnt].Alarm.Link := NOT "AUMA_KP_2_1_DB".AUMA[#ID].Link;
	    #KP[#cnt].Use.Enable := "AUMA_KP_2_1_DB".AUMA[#ID].Use;
	    #KP[#cnt].Name := "AUMA_KP_2_1_DB".AUMA[#ID].Name;
	    #KP[#cnt].Position := INT_TO_REAL("AUMA_KP_2_1_DB".AUMA[#ID].Position) / 10.0;
	    #KP[#cnt].FB.QF := "AUMA_KP_2_1_DB".AUMA[#ID].Message.NotReady;
	    #KP[#cnt].FB.KM_Open := "AUMA_KP_2_1_DB".AUMA[#ID].Message.Opening;
	    #KP[#cnt].FB.KM_Close := "AUMA_KP_2_1_DB".AUMA[#ID].Message.Closing;
	    #KP[#cnt].FB.Open := "AUMA_KP_2_1_DB".AUMA[#ID].Message.Open;
	    #KP[#cnt].FB.Close := "AUMA_KP_2_1_DB".AUMA[#ID].Message.Close;
	    #KP[#cnt]();
	    "AUMA_KP_2_1_DB".AUMA[#ID].Speed := #KP[#cnt].Speed;
	    "AUMA_KP_2_1_DB".AUMA[#ID].CMD.Open := #KP[#cnt].CMD_Open;
	    "AUMA_KP_2_1_DB".AUMA[#ID].CMD.Close := #KP[#cnt].CMD_Close;
	    IF "AUMA_KP_2_1_DB".AUMA[#ID].CMD.Open <> "AUMA_KP_2_1_DB".AUMA[#ID].CMD_last.Open THEN
	        "AUMA_KP_2_1_DB".AUMA[#ID].CMD_last.Open := "AUMA_KP_2_1_DB".AUMA[#ID].CMD.Open;
	        "AUMA_KP_2_1_DB".AUMA[#ID].Update := true;
	    END_IF;
	    IF "AUMA_KP_2_1_DB".AUMA[#ID].CMD.Close <> "AUMA_KP_2_1_DB".AUMA[#ID].CMD_last.Close THEN
	        "AUMA_KP_2_1_DB".AUMA[#ID].CMD_last.Close := "AUMA_KP_2_1_DB".AUMA[#ID].CMD.Close;
	        "AUMA_KP_2_1_DB".AUMA[#ID].Update := true;
	    END_IF;
	END_FOR;
END_FUNCTION_BLOCK

FUNCTION_BLOCK "DRV_AUMA"
{ S7_Optimized_Access := 'FALSE' }
VERSION : 0.1
   VAR 
      CMD { S7_SetPoint := 'False'} : "CMD";   // Блок команд
      Mode : Int;   // Режим работы
      Status : Int;   // Статус устройства
      "FB" : Struct   // Функционал
         QF : Bool;   // Защитный автомат
         KM_Open : Bool;   // Пускатель - открыть
         KM_Close : Bool;   // Пускатель - закрыть
         Open : Bool;   // ОС - открыто
         Close : Bool;   // ОС - закрыто
         Reserv : Bool;
         Local_Open : Bool;   // Локальное открытие
         Local_Close : Bool;   // Локальное закрытие
      END_STRUCT;
      Use : Struct   // Функционал
         QF { S7_SetPoint := 'True'} : Bool;   // Защитный автомат
         KM_Open { S7_SetPoint := 'True'} : Bool;   // Пускатель - открыть
         KM_Close { S7_SetPoint := 'True'} : Bool;   // Пускатель - закрыть
         Open { S7_SetPoint := 'True'} : Bool := true;   // ОС - открыто
         Close { S7_SetPoint := 'True'} : Bool := true;   // ОС - закрыто
         One_KM { S7_SetPoint := 'True'} : Bool;   // Общий пускатель
         Air { S7_SetPoint := 'True'} : Bool;   // пневматика - давить всегда
         Cross { S7_SetPoint := 'True'} : Bool;   // Кросс-замена датчиков
         CMD_Open { S7_SetPoint := 'True'} : Bool := true;
         CMD_Close { S7_SetPoint := 'True'} : Bool;
         CMD_Reset : Bool;
         Local_Keys { S7_SetPoint := 'True'} : Bool;
         Local_EndPoint : Bool := true;
         Enable : Bool;
         CWF { S7_SetPoint := 'True'} : Bool;   // не закрывать при аварии
         Duo : Bool;
      END_STRUCT;
      Alarm : Struct   // Список аварий
         Block : Bool;   // Аварийная остановка
         QF : Bool;   // Выбило защитный автомат
         KM_Open : Bool;   // Не сработал пускатель - открыть
         KM_Close : Bool;   // Не сработал пускатель - закрыть
         Two_S : Bool;   // Две ОС
         Open : Bool;   // Не сработал концевик - открыто
         Close : Bool;   // Не сработал концевик - закрыто
         OpTime : Bool;
         Link : Bool;   // Нет связи
      END_STRUCT;
      support : Word;   // Слово аварий
      CMD_Open : Bool;
      CMD_Close : Bool;
      xON : Bool;
      xOFF : Bool;
      Clock : Array[0..4] of "Time_S";   // Блок таймеров
      CodeID { S7_SetPoint := 'True'} : Int;
      Position : Real;
      Speed { S7_SetPoint := 'True'} : Byte;
      "Name" : String[4];
      PT {InstructionName := 'R_TRIG'; LibVersion := '1.0'; S7_SetPoint := 'False'} : Array[0..1] of R_TRIG;
      NT {InstructionName := 'F_TRIG'; LibVersion := '1.0'; S7_SetPoint := 'False'} : Array[0..1] of F_TRIG;
   END_VAR

   VAR_TEMP 
      dev : Int;
   END_VAR


BEGIN
	//VALVES
	//control of typical air and electrical valves
	// - doors
	// - dampers
	// - valves
	// - etc
	
	//global commands
	//auto mode
	(*
	IF "Reset_Hand" THEN
	    #CMD.Hand := FALSE;
	END_IF;*)
	
	//simulation mode
	#NT[0](CLK := "Sim_All");
	#NT[0](CLK := "Sim_All");
	IF #NT[0].Q THEN
	    #CMD.Sim := TRUE;
	END_IF;
	IF #NT[0].Q THEN
	    #CMD.Sim := FALSE;
	END_IF;
	//global reset
	IF "Reset_All" THEN
	    #CMD.Reset := TRUE;
	END_IF;
	
	//QF control
	IF #FB.QF THEN
	    #Alarm.QF := TRUE;
	END_IF;
	(*
	//KM control
	IF (#CMD_Open AND NOT #xON AND NOT #FB.KM_Open) OR (#CMD_Close AND NOT #xOFF AND NOT #FB.KM_Close) THEN
	    #Clock[0].Start := TRUE;
	    IF #Clock[0]."Exit" AND #CMD_Open THEN
	        #Alarm.KM_Open := TRUE;
	    END_IF;
	    IF #Clock[0]."Exit" AND #CMD_Close THEN
	        #Alarm.KM_Close := TRUE;
	    END_IF;
	ELSE
	    #Clock[0].Start := FALSE;
	END_IF;*)
	
	
	//device control
	"drv_Mode"(CMD := #CMD,
	           All_Block := "All_Block",
	           Mode => #Mode);
	//Hand mode flag
	IF #CMD.Hand THEN
	    "Hand_VD2" := TRUE;
	END_IF;
	
	//delay turn on
	IF #Clock[1].SP > 0 AND NOT #CMD.Hand THEN
	    IF #CMD.Start_M THEN
	        #Clock[1].Start := TRUE;
	        #Clock[2].Start := FALSE;
	        IF #Clock[1]."Exit" THEN
	            #support.%X1 := TRUE;
	        END_IF;
	    ELSE
	        #Clock[1].Start := FALSE;
	    END_IF;
	ELSE
	    #support.%X1 := #CMD.Start_M;
	END_IF;
	
	//delay turn off
	IF #Clock[2].SP > 0 AND NOT #CMD.Hand THEN
	    IF NOT #CMD.Start_M THEN
	        #Clock[1].Start := FALSE;
	        #Clock[2].Start := TRUE;
	        IF #Clock[2]."Exit" THEN
	            #support.%X1 := FALSE;
	        END_IF;
	    ELSE
	        #Clock[2].Start := FALSE;
	    END_IF;
	ELSE
	    #support.%X1 := #CMD.Start_M;
	END_IF;
	
	//Opening
	IF #support.%X1 AND NOT #CMD.Alarm AND NOT #CMD.Sim THEN
	    #support.%X3 := FALSE;
	    IF NOT #FB.Open THEN
	        #support.%X2 := TRUE;
	        #Clock[3].Start := TRUE;
	        #Clock[3].Pause := FALSE;
	    END_IF;
	    #support.%X3 := FALSE;
	    #Clock[4].Start := FALSE;
	    
	    //opening in progress
	    IF NOT #Clock[3]."Exit" AND NOT #FB.Open THEN
	        #Status := 2;
	    END_IF;
	    //opening in fault
	    IF #Clock[3]."Exit" AND NOT #Alarm.Link THEN
	        IF NOT #FB.Open AND NOT #FB.Close THEN
	            #Status := 5;
	        END_IF;
	        IF NOT #FB.Open AND #FB.Close THEN
	            #Status := 7;
	        END_IF;
	        #Alarm.Open := TRUE;
	    END_IF;
	    //opening complieted
	    IF #FB.Open THEN
	        #Status := 1;
	        #Clock[3].Pause := TRUE;
	        #support.%X2 := FALSE;
	        IF #CMD.Alarm THEN
	            #Status := 6;
	            #support.%X2 := FALSE;
	        END_IF;
	    END_IF;
	    
	END_IF;
	
	//Closing
	IF NOT #support.%X1 AND NOT #CMD.Sim THEN
	    #support.%X2 := FALSE;
	    IF NOT #FB.Close THEN
	        #support.%X3 := TRUE;
	        #Clock[4].Start := TRUE;
	        #Clock[4].Pause := FALSE;
	    END_IF;
	    #Clock[3].Start := FALSE;
	    
	    
	    //closing in progress
	    IF NOT #Clock[4]."Exit" AND NOT #FB.Close THEN
	        #Status := 3;
	    END_IF;
	    //closing in fault
	    IF #Clock[4]."Exit" AND NOT #Alarm.Link THEN
	        IF NOT #FB.Close AND NOT #FB.Open THEN
	            #Status := 5;
	        END_IF;
	        IF NOT #FB.Close AND #FB.Open THEN
	            #Status := 6;
	        END_IF;
	        #Alarm.Close := TRUE;
	    END_IF;
	    //closing complieted
	    IF #FB.Close THEN
	        #Status := 0;
	        #Clock[4].Pause := TRUE;
	        #support.%X3 := FALSE;
	        IF #CMD.Alarm THEN
	            #Status := 7;
	            #support.%X3 := FALSE;
	        END_IF;
	    END_IF;
	    
	END_IF;
	
	//alarm control
	IF (#Alarm.Open OR #Alarm.Close OR #Alarm.KM_Close OR #Alarm.KM_Open OR #Alarm.QF(* OR #Alarm.Link*)) AND NOT #CMD.Sim THEN
	    #CMD.Alarm := TRUE;
	    "Alm_VD2" := TRUE;
	END_IF;
	
	//disable close while alarm
	IF #CMD.Alarm THEN
	    #support.%X2 := FALSE;
	    #support.%X3 := FALSE;
	END_IF;
	
	//Simulation
	IF #CMD.Sim THEN
	    IF #support.%X1 THEN
	        #Status := 1;
	    ELSE
	        #Status := 0;
	    END_IF;
	END_IF;
	
	//Local mode
	IF #CMD.Local THEN
	    IF #FB.Open AND NOT #FB.Close THEN
	        #Status := 1;
	    ELSIF NOT #FB.Open AND #FB.Close THEN
	        #Status := 0;
	    ELSE
	        #Status := 2;
	    END_IF;
	    #CMD.Reset := TRUE;
	END_IF;
	
	//ON & OFF
	IF (#FB.Open AND (#CMD.Start_M OR #CMD.Sim)) AND NOT #CMD.Alarm THEN
	    #xON := TRUE;
	    #xOFF := FALSE;
	END_IF;
	IF (#FB.Close AND (NOT #CMD.Start_M OR #CMD.Sim)) AND NOT #CMD.Alarm THEN
	    #xON := FALSE;
	    #xOFF := TRUE;
	END_IF;
	IF (NOT #FB.Close AND NOT #FB.Open) OR #CMD.Alarm THEN
	    #xON := FALSE;
	    #xOFF := FALSE;
	END_IF;
	
	//commands
	//turn on
	IF #support.%X2 THEN
	    #CMD_Open := TRUE;
	    #CMD_Close := FALSE;
	END_IF;
	//turn off
	IF #support.%X3 THEN
	    IF NOT #Use.Duo THEN
	        #CMD_Open := FALSE;
	        #CMD_Close := TRUE;
	    ELSE
	        #CMD_Open := TRUE;
	        #CMD_Close := TRUE;
	    END_IF;
	END_IF;
	
	//shutdown
	IF (NOT #support.%X2 AND NOT #support.%X3) OR #CMD.Sim THEN
	    #CMD_Open := FALSE;
	    #CMD_Close := FALSE;
	END_IF;
	
	//status no connection
	IF #Alarm.Link THEN
	    #Status := 4;
	END_IF;
	
	//reset
	IF #CMD.Reset THEN
	    #Alarm.QF := FALSE;
	    #Alarm.KM_Close := FALSE;
	    #Alarm.KM_Open := FALSE;
	    #Alarm.Close := FALSE;
	    #Alarm.Open := FALSE;
	    #Alarm.Link := FALSE;
	    FOR #dev := 0 TO 4 DO
	        #Clock[#dev].Reset := TRUE;
	    END_FOR;
	    #CMD.Alarm := FALSE;
	    #CMD.Reset := FALSE;
	END_IF;
	
	//call timers
	FOR #dev := 0 TO 4 DO
	    #Clock[#dev]();
	END_FOR;
END_FUNCTION_BLOCK

FUNCTION "Load_KP_2_1" : Void
{ S7_Optimized_Access := 'TRUE' }
VERSION : 0.1
   VAR_IN_OUT 
      ok : Bool;
      load : Int;
      last : Int;
   END_VAR


BEGIN
	//проверка загруженных данных
	IF #load <> #last THEN
	    #ok := FALSE;
	END_IF;
	
	//первичная загрузка данных
	IF NOT #ok THEN
	    "KP_2_1_DB".KP[0].CMD := "KP_2_1_DB".KP[#load].CMD;
	    "KP_2_1_DB".KP[0].Mode := "KP_2_1_DB".KP[#load].Mode;
	    "KP_2_1_DB".KP[0].Status := "KP_2_1_DB".KP[#load].Status;
	    "KP_2_1_DB".KP[0].FB := "KP_2_1_DB".KP[#load].FB;
	    "KP_2_1_DB".KP[0].Use := "KP_2_1_DB".KP[#load].Use;
	    "KP_2_1_DB".KP[0].Alarm := "KP_2_1_DB".KP[#load].Alarm;
	    "KP_2_1_DB".KP[0].Clock[0].SP := "KP_2_1_DB".KP[#load].Clock[0].SP;
	    "KP_2_1_DB".KP[0].Clock[0].Now := "KP_2_1_DB".KP[#load].Clock[0].Now;
	    "KP_2_1_DB".KP[0].Clock[1].SP := "KP_2_1_DB".KP[#load].Clock[1].SP;
	    "KP_2_1_DB".KP[0].Clock[1].Now := "KP_2_1_DB".KP[#load].Clock[1].Now;
	    "KP_2_1_DB".KP[0].Clock[2].SP := "KP_2_1_DB".KP[#load].Clock[2].SP;
	    "KP_2_1_DB".KP[0].Clock[2].Now := "KP_2_1_DB".KP[#load].Clock[2].Now;
	    "KP_2_1_DB".KP[0].Clock[3].SP := "KP_2_1_DB".KP[#load].Clock[3].SP;
	    "KP_2_1_DB".KP[0].Clock[3].Now := "KP_2_1_DB".KP[#load].Clock[3].Now;
	    "KP_2_1_DB".KP[0].Clock[4].SP := "KP_2_1_DB".KP[#load].Clock[4].SP;
	    "KP_2_1_DB".KP[0].Clock[4].Now := "KP_2_1_DB".KP[#load].Clock[4].Now;
	    "KP_2_1_DB".KP[0].CodeID := "KP_2_1_DB".KP[#load].CodeID;
	    "KP_2_1_DB".KP[0].Position := "KP_2_1_DB".KP[#load].Position;
	    "KP_2_1_DB".KP[0].Speed := "KP_2_1_DB".KP[#load].Speed;
	    "KP_2_1_DB".KP[0].Name := "KP_2_1_DB".KP[#load].Name;
	    #ok := true;
	    #last := #load;
	END_IF;
	
	//управление с панели
	IF #ok THEN
	    "KP_2_1_DB".KP[#load].CMD.Hand := "KP_2_1_DB".KP[0].CMD.Hand;
	    "KP_2_1_DB".KP[#load].CMD.Force := "KP_2_1_DB".KP[0].CMD.Force;
	    "KP_2_1_DB".KP[#load].CMD.Start_M := "KP_2_1_DB".KP[0].CMD.Start_M;
	    "KP_2_1_DB".KP[#load].CMD.Reset := "KP_2_1_DB".KP[0].CMD.Reset;
	    "KP_2_1_DB".KP[#load].Use := "KP_2_1_DB".KP[0].Use;
	    "KP_2_1_DB".KP[#load].Clock[0].SP := "KP_2_1_DB".KP[0].Clock[0].SP;
	    "KP_2_1_DB".KP[#load].Clock[1].SP := "KP_2_1_DB".KP[0].Clock[1].SP;
	    "KP_2_1_DB".KP[#load].Clock[2].SP := "KP_2_1_DB".KP[0].Clock[2].SP;
	    "KP_2_1_DB".KP[#load].Clock[3].SP := "KP_2_1_DB".KP[0].Clock[3].SP;
	    "KP_2_1_DB".KP[#load].Clock[4].SP := "KP_2_1_DB".KP[0].Clock[4].SP;
	    "KP_2_1_DB".KP[#load].CodeID := "KP_2_1_DB".KP[0].CodeID;
	    "KP_2_1_DB".KP[#load].Speed := "KP_2_1_DB".KP[0].Speed;
	    "KP_2_1_DB".KP[0].CMD.Local := "KP_2_1_DB".KP[#load].CMD.Local;
	    "KP_2_1_DB".KP[0].CMD.Lock := "KP_2_1_DB".KP[#load].CMD.Lock;
	    "KP_2_1_DB".KP[0].Mode := "KP_2_1_DB".KP[#load].Mode;
	    "KP_2_1_DB".KP[0].Status := "KP_2_1_DB".KP[#load].Status;
	    "KP_2_1_DB".KP[0].FB := "KP_2_1_DB".KP[#load].FB;
	    "KP_2_1_DB".KP[0].Alarm := "KP_2_1_DB".KP[#load].Alarm;
	    "KP_2_1_DB".KP[0].Clock[0].Now := "KP_2_1_DB".KP[#load].Clock[0].Now;
	    "KP_2_1_DB".KP[0].Clock[1].Now := "KP_2_1_DB".KP[#load].Clock[1].Now;
	    "KP_2_1_DB".KP[0].Clock[2].Now := "KP_2_1_DB".KP[#load].Clock[2].Now;
	    "KP_2_1_DB".KP[0].Clock[3].Now := "KP_2_1_DB".KP[#load].Clock[3].Now;
	    "KP_2_1_DB".KP[0].Clock[4].Now := "KP_2_1_DB".KP[#load].Clock[4].Now;
	    "KP_2_1_DB".KP[0].Position := "KP_2_1_DB".KP[#load].Position;
	    IF "KP_2_1_DB".KP[0].CMD.Reset THEN
	        "KP_2_1_DB".KP[0].CMD.Reset := FALSE;
	    END_IF;
	END_IF;
	
	    
END_FUNCTION

FUNCTION_BLOCK "KP_2_2"
{ S7_Optimized_Access := 'FALSE' }
VERSION : 0.1
   VAR 
      limit { S7_SetPoint := 'True'} : Int := 2;   // число задвижек в камере
      load : Int;   // отображаемые на экране настройки
      load_last : Int;
      KP : Array[0..10] of "DRV_AUMA";
      load_ok { S7_SetPoint := 'True'} : Bool;
   END_VAR

   VAR_TEMP 
      ID : Int;
      cnt : Int;
   END_VAR


BEGIN
	//дистанционный режим управления
	FOR #cnt := 1 TO #limit BY 1 DO
	    IF "Comm_SKV_2".To_SKV.Valves.Local[0] THEN
	        IF #KP[#cnt].CMD.Hand THEN
	            #KP[#cnt].CMD.Start_M := "Comm_SKV_2".From_SKV.Valves.REQ[#cnt];
	        END_IF;
	        IF "Comm_SKV_2".From_SKV.Valves.REQ[0] THEN
	            #KP[#cnt].CMD.Reset := TRUE;
	            #load := 10;
	        END_IF;
	    ELSE
	        "Comm_SKV_2".To_SKV.Valves.Local[#cnt] := #KP[#cnt].CMD.Start_M;
	    END_IF;
	END_FOR;
	
	//экранный буфер
	"Load_KP_2_2"(last := #load_last,
	              load := #load,
	              ok := #load_ok);
	IF "KP_Reset" THEN
	    #load := 10;
	END_IF;
	
	FOR #cnt := 1 TO #limit BY 1 DO
	    #ID := #KP[#cnt].CodeID;
	    #KP[#cnt].CMD.Local := NOT "AUMA_KP_2_2_DB".AUMA[#ID].Message.Sel_Dist;
	    #KP[#cnt].Alarm.Link := NOT "AUMA_KP_2_2_DB".AUMA[#ID].Link;
	    #KP[#cnt].Use.Enable := "AUMA_KP_2_2_DB".AUMA[#ID].Use;
	    #KP[#cnt].Name := "AUMA_KP_2_2_DB".AUMA[#ID].Name;
	    #KP[#cnt].Position := INT_TO_REAL("AUMA_KP_2_2_DB".AUMA[#ID].Position) / 10.0;
	    #KP[#cnt].FB.QF := "AUMA_KP_2_2_DB".AUMA[#ID].Message.NotReady;
	    #KP[#cnt].FB.KM_Open := "AUMA_KP_2_2_DB".AUMA[#ID].Message.Opening;
	    #KP[#cnt].FB.KM_Close := "AUMA_KP_2_2_DB".AUMA[#ID].Message.Closing;
	    #KP[#cnt].FB.Open := "AUMA_KP_2_2_DB".AUMA[#ID].Message.Open;
	    #KP[#cnt].FB.Close := "AUMA_KP_2_2_DB".AUMA[#ID].Message.Close;
	    #KP[#cnt]();
	    "AUMA_KP_2_2_DB".AUMA[#ID].Speed := #KP[#cnt].Speed;
	    "AUMA_KP_2_2_DB".AUMA[#ID].CMD.Open := #KP[#cnt].CMD_Open;
	    "AUMA_KP_2_2_DB".AUMA[#ID].CMD.Close := #KP[#cnt].CMD_Close;
	    IF "AUMA_KP_2_2_DB".AUMA[#ID].CMD.Open <> "AUMA_KP_2_2_DB".AUMA[#ID].CMD_last.Open THEN
	        "AUMA_KP_2_2_DB".AUMA[#ID].CMD_last.Open := "AUMA_KP_2_2_DB".AUMA[#ID].CMD.Open;
	        "AUMA_KP_2_2_DB".AUMA[#ID].Update := true;
	    END_IF;
	    IF "AUMA_KP_2_2_DB".AUMA[#ID].CMD.Close <> "AUMA_KP_2_2_DB".AUMA[#ID].CMD_last.Close THEN
	        "AUMA_KP_2_2_DB".AUMA[#ID].CMD_last.Close := "AUMA_KP_2_2_DB".AUMA[#ID].CMD.Close;
	        "AUMA_KP_2_2_DB".AUMA[#ID].Update := true;
	    END_IF;
	END_FOR;
END_FUNCTION_BLOCK

FUNCTION "Load_KP_2_2" : Void
{ S7_Optimized_Access := 'TRUE' }
VERSION : 0.1
   VAR_IN_OUT 
      ok : Bool;
      load : Int;
      last : Int;
   END_VAR


BEGIN
	//проверка загруженных данных
	IF #load <> #last THEN
	    #ok := FALSE;
	END_IF;
	
	//первичная загрузка данных
	IF NOT #ok THEN
	    "KP_2_2_DB".KP[0].CMD := "KP_2_2_DB".KP[#load].CMD;
	    "KP_2_2_DB".KP[0].Mode := "KP_2_2_DB".KP[#load].Mode;
	    "KP_2_2_DB".KP[0].Status := "KP_2_2_DB".KP[#load].Status;
	    "KP_2_2_DB".KP[0].FB := "KP_2_2_DB".KP[#load].FB;
	    "KP_2_2_DB".KP[0].Use := "KP_2_2_DB".KP[#load].Use;
	    "KP_2_2_DB".KP[0].Alarm := "KP_2_2_DB".KP[#load].Alarm;
	    "KP_2_2_DB".KP[0].Clock[0].SP := "KP_2_2_DB".KP[#load].Clock[0].SP;
	    "KP_2_2_DB".KP[0].Clock[0].Now := "KP_2_2_DB".KP[#load].Clock[0].Now;
	    "KP_2_2_DB".KP[0].Clock[1].SP := "KP_2_2_DB".KP[#load].Clock[1].SP;
	    "KP_2_2_DB".KP[0].Clock[1].Now := "KP_2_2_DB".KP[#load].Clock[1].Now;
	    "KP_2_2_DB".KP[0].Clock[2].SP := "KP_2_2_DB".KP[#load].Clock[2].SP;
	    "KP_2_2_DB".KP[0].Clock[2].Now := "KP_2_2_DB".KP[#load].Clock[2].Now;
	    "KP_2_2_DB".KP[0].Clock[3].SP := "KP_2_2_DB".KP[#load].Clock[3].SP;
	    "KP_2_2_DB".KP[0].Clock[3].Now := "KP_2_2_DB".KP[#load].Clock[3].Now;
	    "KP_2_2_DB".KP[0].Clock[4].SP := "KP_2_2_DB".KP[#load].Clock[4].SP;
	    "KP_2_2_DB".KP[0].Clock[4].Now := "KP_2_2_DB".KP[#load].Clock[4].Now;
	    "KP_2_2_DB".KP[0].CodeID := "KP_2_2_DB".KP[#load].CodeID;
	    "KP_2_2_DB".KP[0].Position := "KP_2_2_DB".KP[#load].Position;
	    "KP_2_2_DB".KP[0].Speed := "KP_2_2_DB".KP[#load].Speed;
	    "KP_2_2_DB".KP[0].Name := "KP_2_2_DB".KP[#load].Name;
	    #ok := true;
	    #last := #load;
	END_IF;
	
	//управление с панели
	IF #ok THEN
	    "KP_2_2_DB".KP[#load].CMD.Hand := "KP_2_2_DB".KP[0].CMD.Hand;
	    "KP_2_2_DB".KP[#load].CMD.Force := "KP_2_2_DB".KP[0].CMD.Force;
	    "KP_2_2_DB".KP[#load].CMD.Start_M := "KP_2_2_DB".KP[0].CMD.Start_M;
	    "KP_2_2_DB".KP[#load].CMD.Reset := "KP_2_2_DB".KP[0].CMD.Reset;
	    "KP_2_2_DB".KP[#load].Use := "KP_2_2_DB".KP[0].Use;
	    "KP_2_2_DB".KP[#load].Clock[0].SP := "KP_2_2_DB".KP[0].Clock[0].SP;
	    "KP_2_2_DB".KP[#load].Clock[1].SP := "KP_2_2_DB".KP[0].Clock[1].SP;
	    "KP_2_2_DB".KP[#load].Clock[2].SP := "KP_2_2_DB".KP[0].Clock[2].SP;
	    "KP_2_2_DB".KP[#load].Clock[3].SP := "KP_2_2_DB".KP[0].Clock[3].SP;
	    "KP_2_2_DB".KP[#load].Clock[4].SP := "KP_2_2_DB".KP[0].Clock[4].SP;
	    "KP_2_2_DB".KP[#load].CodeID := "KP_2_2_DB".KP[0].CodeID;
	    "KP_2_2_DB".KP[#load].Speed := "KP_2_2_DB".KP[0].Speed;
	    "KP_2_2_DB".KP[0].CMD.Local := "KP_2_2_DB".KP[#load].CMD.Local;
	    "KP_2_2_DB".KP[0].CMD.Lock := "KP_2_2_DB".KP[#load].CMD.Lock;
	    "KP_2_2_DB".KP[0].Mode := "KP_2_2_DB".KP[#load].Mode;
	    "KP_2_2_DB".KP[0].Status := "KP_2_2_DB".KP[#load].Status;
	    "KP_2_2_DB".KP[0].FB := "KP_2_2_DB".KP[#load].FB;
	    "KP_2_2_DB".KP[0].Alarm := "KP_2_2_DB".KP[#load].Alarm;
	    "KP_2_2_DB".KP[0].Clock[0].Now := "KP_2_2_DB".KP[#load].Clock[0].Now;
	    "KP_2_2_DB".KP[0].Clock[1].Now := "KP_2_2_DB".KP[#load].Clock[1].Now;
	    "KP_2_2_DB".KP[0].Clock[2].Now := "KP_2_2_DB".KP[#load].Clock[2].Now;
	    "KP_2_2_DB".KP[0].Clock[3].Now := "KP_2_2_DB".KP[#load].Clock[3].Now;
	    "KP_2_2_DB".KP[0].Clock[4].Now := "KP_2_2_DB".KP[#load].Clock[4].Now;
	    "KP_2_2_DB".KP[0].Position := "KP_2_2_DB".KP[#load].Position;
	    IF "KP_2_2_DB".KP[0].CMD.Reset THEN
	        "KP_2_2_DB".KP[0].CMD.Reset := FALSE;
	    END_IF;
	END_IF;
	
	    
END_FUNCTION

FUNCTION_BLOCK "KP_2_3"
{ S7_Optimized_Access := 'FALSE' }
VERSION : 0.1
   VAR 
      limit { S7_SetPoint := 'True'} : Int := 2;   // число задвижек в камере
      load : Int;   // отображаемые на экране настройки
      load_last : Int;
      KP : Array[0..10] of "DRV_AUMA";
      load_ok { S7_SetPoint := 'True'} : Bool;
   END_VAR

   VAR_TEMP 
      ID : Int;
      cnt : Int;
   END_VAR


BEGIN
	//дистанционный режим управления
	FOR #cnt := 1 TO #limit BY 1 DO
	    IF "Comm_SKV_20".To_SKV.Valves.Local[0] THEN
	        IF #KP[#cnt].CMD.Hand THEN
	            #KP[#cnt].CMD.Start_M := "Comm_SKV_20".From_SKV.Valves.REQ[#cnt];
	        END_IF;
	        IF "Comm_SKV_20".From_SKV.Valves.REQ[0] THEN
	            #KP[#cnt].CMD.Reset := TRUE;
	            #load := 10;
	        END_IF;
	    ELSE
	        "Comm_SKV_20".To_SKV.Valves.Local[#cnt] := #KP[#cnt].CMD.Start_M;
	    END_IF;
	END_FOR;
	
	//экранный буфер
	"Load_KP_2_3"(last := #load_last,
	              load := #load,
	              ok := #load_ok);
	IF "KP_Reset" THEN
	    #load := 10;
	END_IF;
	
	FOR #cnt := 1 TO #limit BY 1 DO
	    #ID := #KP[#cnt].CodeID;
	    #KP[#cnt].CMD.Local := NOT "AUMA_KP_2_3_DB".AUMA[#ID].Message.Sel_Dist;
	    #KP[#cnt].Alarm.Link := NOT "AUMA_KP_2_3_DB".AUMA[#ID].Link;
	    #KP[#cnt].Use.Enable := "AUMA_KP_2_3_DB".AUMA[#ID].Use;
	    #KP[#cnt].Name := "AUMA_KP_2_3_DB".AUMA[#ID].Name;
	    #KP[#cnt].Position := INT_TO_REAL("AUMA_KP_2_3_DB".AUMA[#ID].Position) / 10.0;
	    #KP[#cnt].FB.QF := "AUMA_KP_2_3_DB".AUMA[#ID].Message.NotReady;
	    #KP[#cnt].FB.KM_Open := "AUMA_KP_2_3_DB".AUMA[#ID].Message.Opening;
	    #KP[#cnt].FB.KM_Close := "AUMA_KP_2_3_DB".AUMA[#ID].Message.Closing;
	    #KP[#cnt].FB.Open := "AUMA_KP_2_3_DB".AUMA[#ID].Message.Open;
	    #KP[#cnt].FB.Close := "AUMA_KP_2_3_DB".AUMA[#ID].Message.Close;
	    #KP[#cnt]();
	    "AUMA_KP_2_3_DB".AUMA[#ID].Speed := #KP[#cnt].Speed;
	    "AUMA_KP_2_3_DB".AUMA[#ID].CMD.Open := #KP[#cnt].CMD_Open;
	    "AUMA_KP_2_3_DB".AUMA[#ID].CMD.Close := #KP[#cnt].CMD_Close;
	    IF "AUMA_KP_2_3_DB".AUMA[#ID].CMD.Open <> "AUMA_KP_2_3_DB".AUMA[#ID].CMD_last.Open THEN
	        "AUMA_KP_2_3_DB".AUMA[#ID].CMD_last.Open := "AUMA_KP_2_3_DB".AUMA[#ID].CMD.Open;
	        "AUMA_KP_2_3_DB".AUMA[#ID].Update := true;
	    END_IF;
	    IF "AUMA_KP_2_3_DB".AUMA[#ID].CMD.Close <> "AUMA_KP_2_3_DB".AUMA[#ID].CMD_last.Close THEN
	        "AUMA_KP_2_3_DB".AUMA[#ID].CMD_last.Close := "AUMA_KP_2_3_DB".AUMA[#ID].CMD.Close;
	        "AUMA_KP_2_3_DB".AUMA[#ID].Update := true;
	    END_IF;
	END_FOR;
END_FUNCTION_BLOCK

FUNCTION "Load_KP_2_3" : Void
{ S7_Optimized_Access := 'TRUE' }
VERSION : 0.1
   VAR_IN_OUT 
      ok : Bool;
      load : Int;
      last : Int;
   END_VAR


BEGIN
	//проверка загруженных данных
	IF #load <> #last THEN
	    #ok := FALSE;
	END_IF;
	
	//первичная загрузка данных
	IF NOT #ok THEN
	    "KP_2_3_DB".KP[0].CMD := "KP_2_3_DB".KP[#load].CMD;
	    "KP_2_3_DB".KP[0].Mode := "KP_2_3_DB".KP[#load].Mode;
	    "KP_2_3_DB".KP[0].Status := "KP_2_3_DB".KP[#load].Status;
	    "KP_2_3_DB".KP[0].FB := "KP_2_3_DB".KP[#load].FB;
	    "KP_2_3_DB".KP[0].Use := "KP_2_3_DB".KP[#load].Use;
	    "KP_2_3_DB".KP[0].Alarm := "KP_2_3_DB".KP[#load].Alarm;
	    "KP_2_3_DB".KP[0].Clock[0].SP := "KP_2_3_DB".KP[#load].Clock[0].SP;
	    "KP_2_3_DB".KP[0].Clock[0].Now := "KP_2_3_DB".KP[#load].Clock[0].Now;
	    "KP_2_3_DB".KP[0].Clock[1].SP := "KP_2_3_DB".KP[#load].Clock[1].SP;
	    "KP_2_3_DB".KP[0].Clock[1].Now := "KP_2_3_DB".KP[#load].Clock[1].Now;
	    "KP_2_3_DB".KP[0].Clock[2].SP := "KP_2_3_DB".KP[#load].Clock[2].SP;
	    "KP_2_3_DB".KP[0].Clock[2].Now := "KP_2_3_DB".KP[#load].Clock[2].Now;
	    "KP_2_3_DB".KP[0].Clock[3].SP := "KP_2_3_DB".KP[#load].Clock[3].SP;
	    "KP_2_3_DB".KP[0].Clock[3].Now := "KP_2_3_DB".KP[#load].Clock[3].Now;
	    "KP_2_3_DB".KP[0].Clock[4].SP := "KP_2_3_DB".KP[#load].Clock[4].SP;
	    "KP_2_3_DB".KP[0].Clock[4].Now := "KP_2_3_DB".KP[#load].Clock[4].Now;
	    "KP_2_3_DB".KP[0].CodeID := "KP_2_3_DB".KP[#load].CodeID;
	    "KP_2_3_DB".KP[0].Position := "KP_2_3_DB".KP[#load].Position;
	    "KP_2_3_DB".KP[0].Speed := "KP_2_3_DB".KP[#load].Speed;
	    "KP_2_3_DB".KP[0].Name := "KP_2_3_DB".KP[#load].Name;
	    #ok := true;
	    #last := #load;
	END_IF;
	
	//управление с панели
	IF #ok THEN
	    "KP_2_3_DB".KP[#load].CMD.Hand := "KP_2_3_DB".KP[0].CMD.Hand;
	    "KP_2_3_DB".KP[#load].CMD.Force := "KP_2_3_DB".KP[0].CMD.Force;
	    "KP_2_3_DB".KP[#load].CMD.Start_M := "KP_2_3_DB".KP[0].CMD.Start_M;
	    "KP_2_3_DB".KP[#load].CMD.Reset := "KP_2_3_DB".KP[0].CMD.Reset;
	    "KP_2_3_DB".KP[#load].Use := "KP_2_3_DB".KP[0].Use;
	    "KP_2_3_DB".KP[#load].Clock[0].SP := "KP_2_3_DB".KP[0].Clock[0].SP;
	    "KP_2_3_DB".KP[#load].Clock[1].SP := "KP_2_3_DB".KP[0].Clock[1].SP;
	    "KP_2_3_DB".KP[#load].Clock[2].SP := "KP_2_3_DB".KP[0].Clock[2].SP;
	    "KP_2_3_DB".KP[#load].Clock[3].SP := "KP_2_3_DB".KP[0].Clock[3].SP;
	    "KP_2_3_DB".KP[#load].Clock[4].SP := "KP_2_3_DB".KP[0].Clock[4].SP;
	    "KP_2_3_DB".KP[#load].CodeID := "KP_2_3_DB".KP[0].CodeID;
	    "KP_2_3_DB".KP[#load].Speed := "KP_2_3_DB".KP[0].Speed;
	    "KP_2_3_DB".KP[0].CMD.Local := "KP_2_3_DB".KP[#load].CMD.Local;
	    "KP_2_3_DB".KP[0].CMD.Lock := "KP_2_3_DB".KP[#load].CMD.Lock;
	    "KP_2_3_DB".KP[0].Mode := "KP_2_3_DB".KP[#load].Mode;
	    "KP_2_3_DB".KP[0].Status := "KP_2_3_DB".KP[#load].Status;
	    "KP_2_3_DB".KP[0].FB := "KP_2_3_DB".KP[#load].FB;
	    "KP_2_3_DB".KP[0].Alarm := "KP_2_3_DB".KP[#load].Alarm;
	    "KP_2_3_DB".KP[0].Clock[0].Now := "KP_2_3_DB".KP[#load].Clock[0].Now;
	    "KP_2_3_DB".KP[0].Clock[1].Now := "KP_2_3_DB".KP[#load].Clock[1].Now;
	    "KP_2_3_DB".KP[0].Clock[2].Now := "KP_2_3_DB".KP[#load].Clock[2].Now;
	    "KP_2_3_DB".KP[0].Clock[3].Now := "KP_2_3_DB".KP[#load].Clock[3].Now;
	    "KP_2_3_DB".KP[0].Clock[4].Now := "KP_2_3_DB".KP[#load].Clock[4].Now;
	    "KP_2_3_DB".KP[0].Position := "KP_2_3_DB".KP[#load].Position;
	    IF "KP_2_3_DB".KP[0].CMD.Reset THEN
	        "KP_2_3_DB".KP[0].CMD.Reset := FALSE;
	    END_IF;
	END_IF;
	
	    
END_FUNCTION

FUNCTION_BLOCK "KP_2_4"
{ S7_Optimized_Access := 'FALSE' }
VERSION : 0.1
   VAR 
      limit { S7_SetPoint := 'True'} : Int := 2;   // число задвижек в камере
      load : Int;   // отображаемые на экране настройки
      load_last : Int;
      KP : Array[0..10] of "DRV_AUMA";
      load_ok { S7_SetPoint := 'True'} : Bool;
   END_VAR

   VAR_TEMP 
      ID : Int;
      cnt : Int;
   END_VAR


BEGIN
	//дистанционный режим управления
	FOR #cnt := 1 TO #limit BY 1 DO
	    IF "Comm_SKV_21".To_SKV.Valves.Local[0] THEN
	        IF #KP[#cnt].CMD.Hand THEN
	            #KP[#cnt].CMD.Start_M := "Comm_SKV_21".From_SKV.Valves.REQ[#cnt];
	        END_IF;
	        IF "Comm_SKV_21".From_SKV.Valves.REQ[0] THEN
	            #KP[#cnt].CMD.Reset := TRUE;
	            #load := 10;
	        END_IF;
	    ELSE
	        "Comm_SKV_21".To_SKV.Valves.Local[#cnt] := #KP[#cnt].CMD.Start_M;
	    END_IF;
	END_FOR;
	
	//экранный буфер
	"Load_KP_2_4"(last := #load_last,
	              load := #load,
	              ok := #load_ok);
	IF "KP_Reset" THEN
	    #load := 10;
	END_IF;
	
	FOR #cnt := 1 TO #limit BY 1 DO
	    #ID := #KP[#cnt].CodeID;
	    #KP[#cnt].CMD.Local := NOT "AUMA_KP_2_4_DB".AUMA[#ID].Message.Sel_Dist;
	    #KP[#cnt].Alarm.Link := NOT "AUMA_KP_2_4_DB".AUMA[#ID].Link;
	    #KP[#cnt].Use.Enable := "AUMA_KP_2_4_DB".AUMA[#ID].Use;
	    #KP[#cnt].Name := "AUMA_KP_2_4_DB".AUMA[#ID].Name;
	    #KP[#cnt].Position := INT_TO_REAL("AUMA_KP_2_4_DB".AUMA[#ID].Position) / 10.0;
	    #KP[#cnt].FB.QF := "AUMA_KP_2_4_DB".AUMA[#ID].Message.NotReady;
	    #KP[#cnt].FB.KM_Open := "AUMA_KP_2_4_DB".AUMA[#ID].Message.Opening;
	    #KP[#cnt].FB.KM_Close := "AUMA_KP_2_4_DB".AUMA[#ID].Message.Closing;
	    #KP[#cnt].FB.Open := "AUMA_KP_2_4_DB".AUMA[#ID].Message.Open;
	    #KP[#cnt].FB.Close := "AUMA_KP_2_4_DB".AUMA[#ID].Message.Close;
	    #KP[#cnt]();
	    "AUMA_KP_2_4_DB".AUMA[#ID].Speed := #KP[#cnt].Speed;
	    "AUMA_KP_2_4_DB".AUMA[#ID].CMD.Open := #KP[#cnt].CMD_Open;
	    "AUMA_KP_2_4_DB".AUMA[#ID].CMD.Close := #KP[#cnt].CMD_Close;
	    IF "AUMA_KP_2_4_DB".AUMA[#ID].CMD.Open <> "AUMA_KP_2_4_DB".AUMA[#ID].CMD_last.Open THEN
	        "AUMA_KP_2_4_DB".AUMA[#ID].CMD_last.Open := "AUMA_KP_2_4_DB".AUMA[#ID].CMD.Open;
	        "AUMA_KP_2_4_DB".AUMA[#ID].Update := true;
	    END_IF;
	    IF "AUMA_KP_2_4_DB".AUMA[#ID].CMD.Close <> "AUMA_KP_2_4_DB".AUMA[#ID].CMD_last.Close THEN
	        "AUMA_KP_2_4_DB".AUMA[#ID].CMD_last.Close := "AUMA_KP_2_4_DB".AUMA[#ID].CMD.Close;
	        "AUMA_KP_2_4_DB".AUMA[#ID].Update := true;
	    END_IF;
	END_FOR;
END_FUNCTION_BLOCK

FUNCTION "Load_KP_2_4" : Void
{ S7_Optimized_Access := 'TRUE' }
VERSION : 0.1
   VAR_IN_OUT 
      ok : Bool;
      load : Int;
      last : Int;
   END_VAR


BEGIN
	//проверка загруженных данных
	IF #load <> #last THEN
	    #ok := FALSE;
	END_IF;
	
	//первичная загрузка данных
	IF NOT #ok THEN
	    "KP_2_4_DB".KP[0].CMD := "KP_2_4_DB".KP[#load].CMD;
	    "KP_2_4_DB".KP[0].Mode := "KP_2_4_DB".KP[#load].Mode;
	    "KP_2_4_DB".KP[0].Status := "KP_2_4_DB".KP[#load].Status;
	    "KP_2_4_DB".KP[0].FB := "KP_2_4_DB".KP[#load].FB;
	    "KP_2_4_DB".KP[0].Use := "KP_2_4_DB".KP[#load].Use;
	    "KP_2_4_DB".KP[0].Alarm := "KP_2_4_DB".KP[#load].Alarm;
	    "KP_2_4_DB".KP[0].Clock[0].SP := "KP_2_4_DB".KP[#load].Clock[0].SP;
	    "KP_2_4_DB".KP[0].Clock[0].Now := "KP_2_4_DB".KP[#load].Clock[0].Now;
	    "KP_2_4_DB".KP[0].Clock[1].SP := "KP_2_4_DB".KP[#load].Clock[1].SP;
	    "KP_2_4_DB".KP[0].Clock[1].Now := "KP_2_4_DB".KP[#load].Clock[1].Now;
	    "KP_2_4_DB".KP[0].Clock[2].SP := "KP_2_4_DB".KP[#load].Clock[2].SP;
	    "KP_2_4_DB".KP[0].Clock[2].Now := "KP_2_4_DB".KP[#load].Clock[2].Now;
	    "KP_2_4_DB".KP[0].Clock[3].SP := "KP_2_4_DB".KP[#load].Clock[3].SP;
	    "KP_2_4_DB".KP[0].Clock[3].Now := "KP_2_4_DB".KP[#load].Clock[3].Now;
	    "KP_2_4_DB".KP[0].Clock[4].SP := "KP_2_4_DB".KP[#load].Clock[4].SP;
	    "KP_2_4_DB".KP[0].Clock[4].Now := "KP_2_4_DB".KP[#load].Clock[4].Now;
	    "KP_2_4_DB".KP[0].CodeID := "KP_2_4_DB".KP[#load].CodeID;
	    "KP_2_4_DB".KP[0].Position := "KP_2_4_DB".KP[#load].Position;
	    "KP_2_4_DB".KP[0].Speed := "KP_2_4_DB".KP[#load].Speed;
	    "KP_2_4_DB".KP[0].Name := "KP_2_4_DB".KP[#load].Name;
	    #ok := true;
	    #last := #load;
	END_IF;
	
	//управление с панели
	IF #ok THEN
	    "KP_2_4_DB".KP[#load].CMD.Hand := "KP_2_4_DB".KP[0].CMD.Hand;
	    "KP_2_4_DB".KP[#load].CMD.Force := "KP_2_4_DB".KP[0].CMD.Force;
	    "KP_2_4_DB".KP[#load].CMD.Start_M := "KP_2_4_DB".KP[0].CMD.Start_M;
	    "KP_2_4_DB".KP[#load].CMD.Reset := "KP_2_4_DB".KP[0].CMD.Reset;
	    "KP_2_4_DB".KP[#load].Use := "KP_2_4_DB".KP[0].Use;
	    "KP_2_4_DB".KP[#load].Clock[0].SP := "KP_2_4_DB".KP[0].Clock[0].SP;
	    "KP_2_4_DB".KP[#load].Clock[1].SP := "KP_2_4_DB".KP[0].Clock[1].SP;
	    "KP_2_4_DB".KP[#load].Clock[2].SP := "KP_2_4_DB".KP[0].Clock[2].SP;
	    "KP_2_4_DB".KP[#load].Clock[3].SP := "KP_2_4_DB".KP[0].Clock[3].SP;
	    "KP_2_4_DB".KP[#load].Clock[4].SP := "KP_2_4_DB".KP[0].Clock[4].SP;
	    "KP_2_4_DB".KP[#load].CodeID := "KP_2_4_DB".KP[0].CodeID;
	    "KP_2_4_DB".KP[#load].Speed := "KP_2_4_DB".KP[0].Speed;
	    "KP_2_4_DB".KP[0].CMD.Local := "KP_2_4_DB".KP[#load].CMD.Local;
	    "KP_2_4_DB".KP[0].CMD.Lock := "KP_2_4_DB".KP[#load].CMD.Lock;
	    "KP_2_4_DB".KP[0].Mode := "KP_2_4_DB".KP[#load].Mode;
	    "KP_2_4_DB".KP[0].Status := "KP_2_4_DB".KP[#load].Status;
	    "KP_2_4_DB".KP[0].FB := "KP_2_4_DB".KP[#load].FB;
	    "KP_2_4_DB".KP[0].Alarm := "KP_2_4_DB".KP[#load].Alarm;
	    "KP_2_4_DB".KP[0].Clock[0].Now := "KP_2_4_DB".KP[#load].Clock[0].Now;
	    "KP_2_4_DB".KP[0].Clock[1].Now := "KP_2_4_DB".KP[#load].Clock[1].Now;
	    "KP_2_4_DB".KP[0].Clock[2].Now := "KP_2_4_DB".KP[#load].Clock[2].Now;
	    "KP_2_4_DB".KP[0].Clock[3].Now := "KP_2_4_DB".KP[#load].Clock[3].Now;
	    "KP_2_4_DB".KP[0].Clock[4].Now := "KP_2_4_DB".KP[#load].Clock[4].Now;
	    "KP_2_4_DB".KP[0].Position := "KP_2_4_DB".KP[#load].Position;
	    IF "KP_2_4_DB".KP[0].CMD.Reset THEN
	        "KP_2_4_DB".KP[0].CMD.Reset := FALSE;
	    END_IF;
	    END_IF;
	
	    
END_FUNCTION

FUNCTION_BLOCK "KP_2_5"
{ S7_Optimized_Access := 'FALSE' }
VERSION : 0.1
   VAR 
      limit { S7_SetPoint := 'True'} : Int := 2;   // число задвижек в камере
      load : Int;   // отображаемые на экране настройки
      load_last : Int;
      KP : Array[0..10] of "DRV_AUMA";
      load_ok { S7_SetPoint := 'True'} : Bool;
   END_VAR

   VAR_TEMP 
      ID : Int;
      cnt : Int;
   END_VAR


BEGIN
	//дистанционный режим управления
	FOR #cnt := 1 TO #limit BY 1 DO
	    IF "Comm_SKV_22".To_SKV.Valves.Local[0] THEN
	        IF #KP[#cnt].CMD.Hand THEN
	            #KP[#cnt].CMD.Start_M := "Comm_SKV_22".From_SKV.Valves.REQ[#cnt];
	        END_IF;
	        IF "Comm_SKV_22".From_SKV.Valves.REQ[0] THEN
	            #KP[#cnt].CMD.Reset := TRUE;
	            #load := 10;
	        END_IF;
	    ELSE
	        "Comm_SKV_22".To_SKV.Valves.Local[#cnt] := #KP[#cnt].CMD.Start_M;
	    END_IF;
	END_FOR;
	
	//экранный буфер
	"Load_KP_2_5"(last := #load_last,
	              load := #load,
	              ok := #load_ok);
	IF "KP_Reset" THEN
	    #load := 10;
	END_IF;
	
	FOR #cnt := 1 TO #limit BY 1 DO
	    #ID := #KP[#cnt].CodeID;
	    #KP[#cnt].CMD.Local := NOT "AUMA_KP_2_5_DB".AUMA[#ID].Message.Sel_Dist;
	    #KP[#cnt].Alarm.Link := NOT "AUMA_KP_2_5_DB".AUMA[#ID].Link;
	    #KP[#cnt].Use.Enable := "AUMA_KP_2_5_DB".AUMA[#ID].Use;
	    #KP[#cnt].Name := "AUMA_KP_2_5_DB".AUMA[#ID].Name;
	    #KP[#cnt].Position := INT_TO_REAL("AUMA_KP_2_5_DB".AUMA[#ID].Position) / 10.0;
	    #KP[#cnt].FB.QF := "AUMA_KP_2_5_DB".AUMA[#ID].Message.NotReady;
	    #KP[#cnt].FB.KM_Open := "AUMA_KP_2_5_DB".AUMA[#ID].Message.Opening;
	    #KP[#cnt].FB.KM_Close := "AUMA_KP_2_5_DB".AUMA[#ID].Message.Closing;
	    #KP[#cnt].FB.Open := "AUMA_KP_2_5_DB".AUMA[#ID].Message.Open;
	    #KP[#cnt].FB.Close := "AUMA_KP_2_5_DB".AUMA[#ID].Message.Close;
	    #KP[#cnt]();
	    "AUMA_KP_2_5_DB".AUMA[#ID].Speed := #KP[#cnt].Speed;
	    "AUMA_KP_2_5_DB".AUMA[#ID].CMD.Open := #KP[#cnt].CMD_Open;
	    "AUMA_KP_2_5_DB".AUMA[#ID].CMD.Close := #KP[#cnt].CMD_Close;
	    IF "AUMA_KP_2_5_DB".AUMA[#ID].CMD.Open <> "AUMA_KP_2_5_DB".AUMA[#ID].CMD_last.Open THEN
	        "AUMA_KP_2_5_DB".AUMA[#ID].CMD_last.Open := "AUMA_KP_2_5_DB".AUMA[#ID].CMD.Open;
	        "AUMA_KP_2_5_DB".AUMA[#ID].Update := true;
	    END_IF;
	    IF "AUMA_KP_2_5_DB".AUMA[#ID].CMD.Close <> "AUMA_KP_2_5_DB".AUMA[#ID].CMD_last.Close THEN
	        "AUMA_KP_2_5_DB".AUMA[#ID].CMD_last.Close := "AUMA_KP_2_5_DB".AUMA[#ID].CMD.Close;
	        "AUMA_KP_2_5_DB".AUMA[#ID].Update := true;
	    END_IF;
	END_FOR;
END_FUNCTION_BLOCK

FUNCTION "Load_KP_2_5" : Void
{ S7_Optimized_Access := 'TRUE' }
VERSION : 0.1
   VAR_IN_OUT 
      ok : Bool;
      load : Int;
      last : Int;
   END_VAR


BEGIN
	//проверка загруженных данных
	IF #load <> #last THEN
	    #ok := FALSE;
	END_IF;
	
	//первичная загрузка данных
	IF NOT #ok THEN
	    "KP_2_5_DB".KP[0].CMD := "KP_2_5_DB".KP[#load].CMD;
	    "KP_2_5_DB".KP[0].Mode := "KP_2_5_DB".KP[#load].Mode;
	    "KP_2_5_DB".KP[0].Status := "KP_2_5_DB".KP[#load].Status;
	    "KP_2_5_DB".KP[0].FB := "KP_2_5_DB".KP[#load].FB;
	    "KP_2_5_DB".KP[0].Use := "KP_2_5_DB".KP[#load].Use;
	    "KP_2_5_DB".KP[0].Alarm := "KP_2_5_DB".KP[#load].Alarm;
	    "KP_2_5_DB".KP[0].Clock[0].SP := "KP_2_5_DB".KP[#load].Clock[0].SP;
	    "KP_2_5_DB".KP[0].Clock[0].Now := "KP_2_5_DB".KP[#load].Clock[0].Now;
	    "KP_2_5_DB".KP[0].Clock[1].SP := "KP_2_5_DB".KP[#load].Clock[1].SP;
	    "KP_2_5_DB".KP[0].Clock[1].Now := "KP_2_5_DB".KP[#load].Clock[1].Now;
	    "KP_2_5_DB".KP[0].Clock[2].SP := "KP_2_5_DB".KP[#load].Clock[2].SP;
	    "KP_2_5_DB".KP[0].Clock[2].Now := "KP_2_5_DB".KP[#load].Clock[2].Now;
	    "KP_2_5_DB".KP[0].Clock[3].SP := "KP_2_5_DB".KP[#load].Clock[3].SP;
	    "KP_2_5_DB".KP[0].Clock[3].Now := "KP_2_5_DB".KP[#load].Clock[3].Now;
	    "KP_2_5_DB".KP[0].Clock[4].SP := "KP_2_5_DB".KP[#load].Clock[4].SP;
	    "KP_2_5_DB".KP[0].Clock[4].Now := "KP_2_5_DB".KP[#load].Clock[4].Now;
	    "KP_2_5_DB".KP[0].CodeID := "KP_2_5_DB".KP[#load].CodeID;
	    "KP_2_5_DB".KP[0].Position := "KP_2_5_DB".KP[#load].Position;
	    "KP_2_5_DB".KP[0].Speed := "KP_2_5_DB".KP[#load].Speed;
	    "KP_2_5_DB".KP[0].Name := "KP_2_5_DB".KP[#load].Name;
	    #ok := true;
	    #last := #load;
	END_IF;
	
	//управление с панели
	IF #ok THEN
	    "KP_2_5_DB".KP[#load].CMD.Hand := "KP_2_5_DB".KP[0].CMD.Hand;
	    "KP_2_5_DB".KP[#load].CMD.Force := "KP_2_5_DB".KP[0].CMD.Force;
	    "KP_2_5_DB".KP[#load].CMD.Start_M := "KP_2_5_DB".KP[0].CMD.Start_M;
	    "KP_2_5_DB".KP[#load].CMD.Reset := "KP_2_5_DB".KP[0].CMD.Reset;
	    "KP_2_5_DB".KP[#load].Use := "KP_2_5_DB".KP[0].Use;
	    "KP_2_5_DB".KP[#load].Clock[0].SP := "KP_2_5_DB".KP[0].Clock[0].SP;
	    "KP_2_5_DB".KP[#load].Clock[1].SP := "KP_2_5_DB".KP[0].Clock[1].SP;
	    "KP_2_5_DB".KP[#load].Clock[2].SP := "KP_2_5_DB".KP[0].Clock[2].SP;
	    "KP_2_5_DB".KP[#load].Clock[3].SP := "KP_2_5_DB".KP[0].Clock[3].SP;
	    "KP_2_5_DB".KP[#load].Clock[4].SP := "KP_2_5_DB".KP[0].Clock[4].SP;
	    "KP_2_5_DB".KP[#load].CodeID := "KP_2_5_DB".KP[0].CodeID;
	    "KP_2_5_DB".KP[#load].Speed := "KP_2_5_DB".KP[0].Speed;
	    "KP_2_5_DB".KP[0].CMD.Local := "KP_2_5_DB".KP[#load].CMD.Local;
	    "KP_2_5_DB".KP[0].CMD.Lock := "KP_2_5_DB".KP[#load].CMD.Lock;
	    "KP_2_5_DB".KP[0].Mode := "KP_2_5_DB".KP[#load].Mode;
	    "KP_2_5_DB".KP[0].Status := "KP_2_5_DB".KP[#load].Status;
	    "KP_2_5_DB".KP[0].FB := "KP_2_5_DB".KP[#load].FB;
	    "KP_2_5_DB".KP[0].Alarm := "KP_2_5_DB".KP[#load].Alarm;
	    "KP_2_5_DB".KP[0].Clock[0].Now := "KP_2_5_DB".KP[#load].Clock[0].Now;
	    "KP_2_5_DB".KP[0].Clock[1].Now := "KP_2_5_DB".KP[#load].Clock[1].Now;
	    "KP_2_5_DB".KP[0].Clock[2].Now := "KP_2_5_DB".KP[#load].Clock[2].Now;
	    "KP_2_5_DB".KP[0].Clock[3].Now := "KP_2_5_DB".KP[#load].Clock[3].Now;
	    "KP_2_5_DB".KP[0].Clock[4].Now := "KP_2_5_DB".KP[#load].Clock[4].Now;
	    "KP_2_5_DB".KP[0].Position := "KP_2_5_DB".KP[#load].Position;
	    IF "KP_2_5_DB".KP[0].CMD.Reset THEN
	        "KP_2_5_DB".KP[0].CMD.Reset := FALSE;
	    END_IF;
	END_IF;
	
	    
END_FUNCTION

FUNCTION_BLOCK "KP_2_6"
{ S7_Optimized_Access := 'FALSE' }
VERSION : 0.1
   VAR 
      limit { S7_SetPoint := 'True'} : Int := 2;   // число задвижек в камере
      load : Int;   // отображаемые на экране настройки
      load_last : Int;
      KP : Array[0..10] of "DRV_AUMA";
      load_ok { S7_SetPoint := 'True'} : Bool;
   END_VAR

   VAR_TEMP 
      ID : Int;
      cnt : Int;
   END_VAR


BEGIN
	//дистанционный режим управления
	FOR #cnt := 1 TO #limit BY 1 DO
	    IF "Comm_SKV_14".To_SKV.Valves.Local[0] THEN
	        IF #KP[#cnt].CMD.Hand THEN
	            #KP[#cnt].CMD.Start_M := "Comm_SKV_14".From_SKV.Valves.REQ[#cnt];
	        END_IF;
	        IF "Comm_SKV_14".From_SKV.Valves.REQ[0] THEN
	            #KP[#cnt].CMD.Reset := TRUE;
	            #load := 10;
	        END_IF;
	    ELSE
	        "Comm_SKV_14".To_SKV.Valves.Local[#cnt] := #KP[#cnt].CMD.Start_M;
	    END_IF;
	END_FOR;
	
	//экранный буфер
	"Load_KP_2_6"(last := #load_last,
	              load := #load,
	              ok := #load_ok);
	IF "KP_Reset" THEN
	    #load := 10;
	END_IF;
	
	FOR #cnt := 1 TO #limit BY 1 DO
	    #ID := #KP[#cnt].CodeID;
	    #KP[#cnt].CMD.Local := NOT "AUMA_KP_2_6_DB".AUMA[#ID].Message.Sel_Dist;
	    #KP[#cnt].Alarm.Link := NOT "AUMA_KP_2_6_DB".AUMA[#ID].Link;
	    #KP[#cnt].Use.Enable := "AUMA_KP_2_6_DB".AUMA[#ID].Use;
	    #KP[#cnt].Name := "AUMA_KP_2_6_DB".AUMA[#ID].Name;
	    #KP[#cnt].Position := INT_TO_REAL("AUMA_KP_2_6_DB".AUMA[#ID].Position) / 10.0;
	    #KP[#cnt].FB.QF := "AUMA_KP_2_6_DB".AUMA[#ID].Message.NotReady;
	    #KP[#cnt].FB.KM_Open := "AUMA_KP_2_6_DB".AUMA[#ID].Message.Opening;
	    #KP[#cnt].FB.KM_Close := "AUMA_KP_2_6_DB".AUMA[#ID].Message.Closing;
	    #KP[#cnt].FB.Open := "AUMA_KP_2_6_DB".AUMA[#ID].Message.Open;
	    #KP[#cnt].FB.Close := "AUMA_KP_2_6_DB".AUMA[#ID].Message.Close;
	    #KP[#cnt]();
	    "AUMA_KP_2_6_DB".AUMA[#ID].Speed := #KP[#cnt].Speed;
	    "AUMA_KP_2_6_DB".AUMA[#ID].CMD.Open := #KP[#cnt].CMD_Open;
	    "AUMA_KP_2_6_DB".AUMA[#ID].CMD.Close := #KP[#cnt].CMD_Close;
	    IF "AUMA_KP_2_6_DB".AUMA[#ID].CMD.Open <> "AUMA_KP_2_6_DB".AUMA[#ID].CMD_last.Open THEN
	        "AUMA_KP_2_6_DB".AUMA[#ID].CMD_last.Open := "AUMA_KP_2_6_DB".AUMA[#ID].CMD.Open;
	        "AUMA_KP_2_6_DB".AUMA[#ID].Update := true;
	    END_IF;
	    IF "AUMA_KP_2_6_DB".AUMA[#ID].CMD.Close <> "AUMA_KP_2_6_DB".AUMA[#ID].CMD_last.Close THEN
	        "AUMA_KP_2_6_DB".AUMA[#ID].CMD_last.Close := "AUMA_KP_2_6_DB".AUMA[#ID].CMD.Close;
	        "AUMA_KP_2_6_DB".AUMA[#ID].Update := true;
	    END_IF;
	END_FOR;
END_FUNCTION_BLOCK

FUNCTION "Load_KP_2_6" : Void
{ S7_Optimized_Access := 'TRUE' }
VERSION : 0.1
   VAR_IN_OUT 
      ok : Bool;
      load : Int;
      last : Int;
   END_VAR


BEGIN
	//проверка загруженных данных
	IF #load <> #last THEN
	    #ok := FALSE;
	END_IF;
	
	//первичная загрузка данных
	IF NOT #ok THEN
	    "KP_2_6_DB".KP[0].CMD := "KP_2_6_DB".KP[#load].CMD;
	    "KP_2_6_DB".KP[0].Mode := "KP_2_6_DB".KP[#load].Mode;
	    "KP_2_6_DB".KP[0].Status := "KP_2_6_DB".KP[#load].Status;
	    "KP_2_6_DB".KP[0].FB := "KP_2_6_DB".KP[#load].FB;
	    "KP_2_6_DB".KP[0].Use := "KP_2_6_DB".KP[#load].Use;
	    "KP_2_6_DB".KP[0].Alarm := "KP_2_6_DB".KP[#load].Alarm;
	    "KP_2_6_DB".KP[0].Clock[0].SP := "KP_2_6_DB".KP[#load].Clock[0].SP;
	    "KP_2_6_DB".KP[0].Clock[0].Now := "KP_2_6_DB".KP[#load].Clock[0].Now;
	    "KP_2_6_DB".KP[0].Clock[1].SP := "KP_2_6_DB".KP[#load].Clock[1].SP;
	    "KP_2_6_DB".KP[0].Clock[1].Now := "KP_2_6_DB".KP[#load].Clock[1].Now;
	    "KP_2_6_DB".KP[0].Clock[2].SP := "KP_2_6_DB".KP[#load].Clock[2].SP;
	    "KP_2_6_DB".KP[0].Clock[2].Now := "KP_2_6_DB".KP[#load].Clock[2].Now;
	    "KP_2_6_DB".KP[0].Clock[3].SP := "KP_2_6_DB".KP[#load].Clock[3].SP;
	    "KP_2_6_DB".KP[0].Clock[3].Now := "KP_2_6_DB".KP[#load].Clock[3].Now;
	    "KP_2_6_DB".KP[0].Clock[4].SP := "KP_2_6_DB".KP[#load].Clock[4].SP;
	    "KP_2_6_DB".KP[0].Clock[4].Now := "KP_2_6_DB".KP[#load].Clock[4].Now;
	    "KP_2_6_DB".KP[0].CodeID := "KP_2_6_DB".KP[#load].CodeID;
	    "KP_2_6_DB".KP[0].Position := "KP_2_6_DB".KP[#load].Position;
	    "KP_2_6_DB".KP[0].Speed := "KP_2_6_DB".KP[#load].Speed;
	    "KP_2_6_DB".KP[0].Name := "KP_2_6_DB".KP[#load].Name;
	    #ok := true;
	    #last := #load;
	END_IF;
	
	//управление с панели
	IF #ok THEN
	    "KP_2_6_DB".KP[#load].CMD.Hand := "KP_2_6_DB".KP[0].CMD.Hand;
	    "KP_2_6_DB".KP[#load].CMD.Force := "KP_2_6_DB".KP[0].CMD.Force;
	    "KP_2_6_DB".KP[#load].CMD.Start_M := "KP_2_6_DB".KP[0].CMD.Start_M;
	    "KP_2_6_DB".KP[#load].CMD.Reset := "KP_2_6_DB".KP[0].CMD.Reset;
	    "KP_2_6_DB".KP[#load].Use := "KP_2_6_DB".KP[0].Use;
	    "KP_2_6_DB".KP[#load].Clock[0].SP := "KP_2_6_DB".KP[0].Clock[0].SP;
	    "KP_2_6_DB".KP[#load].Clock[1].SP := "KP_2_6_DB".KP[0].Clock[1].SP;
	    "KP_2_6_DB".KP[#load].Clock[2].SP := "KP_2_6_DB".KP[0].Clock[2].SP;
	    "KP_2_6_DB".KP[#load].Clock[3].SP := "KP_2_6_DB".KP[0].Clock[3].SP;
	    "KP_2_6_DB".KP[#load].Clock[4].SP := "KP_2_6_DB".KP[0].Clock[4].SP;
	    "KP_2_6_DB".KP[#load].CodeID := "KP_2_6_DB".KP[0].CodeID;
	    "KP_2_6_DB".KP[#load].Speed := "KP_2_6_DB".KP[0].Speed;
	    "KP_2_6_DB".KP[0].CMD.Local := "KP_2_6_DB".KP[#load].CMD.Local;
	    "KP_2_6_DB".KP[0].CMD.Lock := "KP_2_6_DB".KP[#load].CMD.Lock;
	    "KP_2_6_DB".KP[0].Mode := "KP_2_6_DB".KP[#load].Mode;
	    "KP_2_6_DB".KP[0].Status := "KP_2_6_DB".KP[#load].Status;
	    "KP_2_6_DB".KP[0].FB := "KP_2_6_DB".KP[#load].FB;
	    "KP_2_6_DB".KP[0].Alarm := "KP_2_6_DB".KP[#load].Alarm;
	    "KP_2_6_DB".KP[0].Clock[0].Now := "KP_2_6_DB".KP[#load].Clock[0].Now;
	    "KP_2_6_DB".KP[0].Clock[1].Now := "KP_2_6_DB".KP[#load].Clock[1].Now;
	    "KP_2_6_DB".KP[0].Clock[2].Now := "KP_2_6_DB".KP[#load].Clock[2].Now;
	    "KP_2_6_DB".KP[0].Clock[3].Now := "KP_2_6_DB".KP[#load].Clock[3].Now;
	    "KP_2_6_DB".KP[0].Clock[4].Now := "KP_2_6_DB".KP[#load].Clock[4].Now;
	    "KP_2_6_DB".KP[0].Position := "KP_2_6_DB".KP[#load].Position;
	    IF "KP_2_6_DB".KP[0].CMD.Reset THEN
	        "KP_2_6_DB".KP[0].CMD.Reset := FALSE;
	    END_IF;
	END_IF;
	
	    
END_FUNCTION

FUNCTION_BLOCK "KP_2_7"
{ S7_Optimized_Access := 'FALSE' }
VERSION : 0.1
   VAR 
      limit { S7_SetPoint := 'True'} : Int := 2;   // число задвижек в камере
      load : Int;   // отображаемые на экране настройки
      load_last : Int;
      KP : Array[0..10] of "DRV_AUMA";
      load_ok { S7_SetPoint := 'True'} : Bool;
   END_VAR

   VAR_TEMP 
      ID : Int;
      cnt : Int;
   END_VAR


BEGIN
	//дистанционный режим управления
	FOR #cnt := 1 TO #limit BY 1 DO
	    IF "Comm_SKV_13".To_SKV.Valves.Local[0] THEN
	        IF #KP[#cnt].CMD.Hand THEN
	            #KP[#cnt].CMD.Start_M := "Comm_SKV_13".From_SKV.Valves.REQ[#cnt];
	        END_IF;
	        IF "Comm_SKV_13".From_SKV.Valves.REQ[0] THEN
	            #KP[#cnt].CMD.Reset := TRUE;
	            #load := 10;
	        END_IF;
	    ELSE
	        "Comm_SKV_13".To_SKV.Valves.Local[#cnt] := #KP[#cnt].CMD.Start_M;
	    END_IF;
	END_FOR;
	    
	//экранный буфер
	"Load_KP_2_7"(last := #load_last,
	              load := #load,
	              ok := #load_ok);
	IF "KP_Reset" THEN
	    #load := 10;
	END_IF;
	
	//проброс данных и вызов на исполнение
	FOR #cnt := 1 TO #limit BY 1 DO
	    #ID := #KP[#cnt].CodeID;
	    #KP[#cnt].CMD.Local := NOT "AUMA_KP_2_7_DB".AUMA[#ID].Message.Sel_Dist;
	    #KP[#cnt].Alarm.Link := NOT "AUMA_KP_2_7_DB".AUMA[#ID].Link;
	    #KP[#cnt].Use.Enable := "AUMA_KP_2_7_DB".AUMA[#ID].Use;
	    #KP[#cnt].Name := "AUMA_KP_2_7_DB".AUMA[#ID].Name;
	    #KP[#cnt].Position := INT_TO_REAL("AUMA_KP_2_7_DB".AUMA[#ID].Position) / 10.0;
	    #KP[#cnt].FB.QF := "AUMA_KP_2_7_DB".AUMA[#ID].Message.NotReady;
	    #KP[#cnt].FB.KM_Open := "AUMA_KP_2_7_DB".AUMA[#ID].Message.Opening;
	    #KP[#cnt].FB.KM_Close := "AUMA_KP_2_7_DB".AUMA[#ID].Message.Closing;
	    #KP[#cnt].FB.Open := "AUMA_KP_2_7_DB".AUMA[#ID].Message.Open;
	    #KP[#cnt].FB.Close := "AUMA_KP_2_7_DB".AUMA[#ID].Message.Close;
	    #KP[#cnt]();
	    "AUMA_KP_2_7_DB".AUMA[#ID].Speed := #KP[#cnt].Speed;
	    "AUMA_KP_2_7_DB".AUMA[#ID].CMD.Open := #KP[#cnt].CMD_Open;
	    "AUMA_KP_2_7_DB".AUMA[#ID].CMD.Close := #KP[#cnt].CMD_Close;
	    IF "AUMA_KP_2_7_DB".AUMA[#ID].CMD.Open <> "AUMA_KP_2_7_DB".AUMA[#ID].CMD_last.Open THEN
	        "AUMA_KP_2_7_DB".AUMA[#ID].CMD_last.Open := "AUMA_KP_2_7_DB".AUMA[#ID].CMD.Open;
	        "AUMA_KP_2_7_DB".AUMA[#ID].Update := true;
	    END_IF;
	    IF "AUMA_KP_2_7_DB".AUMA[#ID].CMD.Close <> "AUMA_KP_2_7_DB".AUMA[#ID].CMD_last.Close THEN
	        "AUMA_KP_2_7_DB".AUMA[#ID].CMD_last.Close := "AUMA_KP_2_7_DB".AUMA[#ID].CMD.Close;
	        "AUMA_KP_2_7_DB".AUMA[#ID].Update := true;
	    END_IF;
	END_FOR;
END_FUNCTION_BLOCK

FUNCTION "Load_KP_2_7" : Void
{ S7_Optimized_Access := 'TRUE' }
VERSION : 0.1
   VAR_IN_OUT 
      ok : Bool;
      load : Int;
      last : Int;
   END_VAR


BEGIN
	//проверка загруженных данных
	IF #load <> #last THEN
	    #ok := FALSE;
	END_IF;
	
	//первичная загрузка данных
	IF NOT #ok THEN
	    "KP_2_7_DB".KP[0].CMD := "KP_2_7_DB".KP[#load].CMD;
	    "KP_2_7_DB".KP[0].Mode := "KP_2_7_DB".KP[#load].Mode;
	    "KP_2_7_DB".KP[0].Status := "KP_2_7_DB".KP[#load].Status;
	    "KP_2_7_DB".KP[0].FB := "KP_2_7_DB".KP[#load].FB;
	    "KP_2_7_DB".KP[0].Use := "KP_2_7_DB".KP[#load].Use;
	    "KP_2_7_DB".KP[0].Alarm := "KP_2_7_DB".KP[#load].Alarm;
	    "KP_2_7_DB".KP[0].Clock[0].SP := "KP_2_7_DB".KP[#load].Clock[0].SP;
	    "KP_2_7_DB".KP[0].Clock[0].Now := "KP_2_7_DB".KP[#load].Clock[0].Now;
	    "KP_2_7_DB".KP[0].Clock[1].SP := "KP_2_7_DB".KP[#load].Clock[1].SP;
	    "KP_2_7_DB".KP[0].Clock[1].Now := "KP_2_7_DB".KP[#load].Clock[1].Now;
	    "KP_2_7_DB".KP[0].Clock[2].SP := "KP_2_7_DB".KP[#load].Clock[2].SP;
	    "KP_2_7_DB".KP[0].Clock[2].Now := "KP_2_7_DB".KP[#load].Clock[2].Now;
	    "KP_2_7_DB".KP[0].Clock[3].SP := "KP_2_7_DB".KP[#load].Clock[3].SP;
	    "KP_2_7_DB".KP[0].Clock[3].Now := "KP_2_7_DB".KP[#load].Clock[3].Now;
	    "KP_2_7_DB".KP[0].Clock[4].SP := "KP_2_7_DB".KP[#load].Clock[4].SP;
	    "KP_2_7_DB".KP[0].Clock[4].Now := "KP_2_7_DB".KP[#load].Clock[4].Now;
	    "KP_2_7_DB".KP[0].CodeID := "KP_2_7_DB".KP[#load].CodeID;
	    "KP_2_7_DB".KP[0].Position := "KP_2_7_DB".KP[#load].Position;
	    "KP_2_7_DB".KP[0].Speed := "KP_2_7_DB".KP[#load].Speed;
	    "KP_2_7_DB".KP[0].Name := "KP_2_7_DB".KP[#load].Name;
	    #ok := true;
	    #last := #load;
	END_IF;
	
	//управление с панели
	IF #ok THEN
	    "KP_2_7_DB".KP[#load].CMD.Hand := "KP_2_7_DB".KP[0].CMD.Hand;
	    "KP_2_7_DB".KP[#load].CMD.Force := "KP_2_7_DB".KP[0].CMD.Force;
	    "KP_2_7_DB".KP[#load].CMD.Start_M := "KP_2_7_DB".KP[0].CMD.Start_M;
	    "KP_2_7_DB".KP[#load].CMD.Reset := "KP_2_7_DB".KP[0].CMD.Reset;
	    "KP_2_7_DB".KP[#load].Use := "KP_2_7_DB".KP[0].Use;
	    "KP_2_7_DB".KP[#load].Clock[0].SP := "KP_2_7_DB".KP[0].Clock[0].SP;
	    "KP_2_7_DB".KP[#load].Clock[1].SP := "KP_2_7_DB".KP[0].Clock[1].SP;
	    "KP_2_7_DB".KP[#load].Clock[2].SP := "KP_2_7_DB".KP[0].Clock[2].SP;
	    "KP_2_7_DB".KP[#load].Clock[3].SP := "KP_2_7_DB".KP[0].Clock[3].SP;
	    "KP_2_7_DB".KP[#load].Clock[4].SP := "KP_2_7_DB".KP[0].Clock[4].SP;
	    "KP_2_7_DB".KP[#load].CodeID := "KP_2_7_DB".KP[0].CodeID;
	    "KP_2_7_DB".KP[#load].Speed := "KP_2_7_DB".KP[0].Speed;
	    "KP_2_7_DB".KP[0].CMD.Local := "KP_2_7_DB".KP[#load].CMD.Local;
	    "KP_2_7_DB".KP[0].CMD.Lock := "KP_2_7_DB".KP[#load].CMD.Lock;
	    "KP_2_7_DB".KP[0].Mode := "KP_2_7_DB".KP[#load].Mode;
	    "KP_2_7_DB".KP[0].Status := "KP_2_7_DB".KP[#load].Status;
	    "KP_2_7_DB".KP[0].FB := "KP_2_7_DB".KP[#load].FB;
	    "KP_2_7_DB".KP[0].Alarm := "KP_2_7_DB".KP[#load].Alarm;
	    "KP_2_7_DB".KP[0].Clock[0].Now := "KP_2_7_DB".KP[#load].Clock[0].Now;
	    "KP_2_7_DB".KP[0].Clock[1].Now := "KP_2_7_DB".KP[#load].Clock[1].Now;
	    "KP_2_7_DB".KP[0].Clock[2].Now := "KP_2_7_DB".KP[#load].Clock[2].Now;
	    "KP_2_7_DB".KP[0].Clock[3].Now := "KP_2_7_DB".KP[#load].Clock[3].Now;
	    "KP_2_7_DB".KP[0].Clock[4].Now := "KP_2_7_DB".KP[#load].Clock[4].Now;
	    "KP_2_7_DB".KP[0].Position := "KP_2_7_DB".KP[#load].Position;
	    IF "KP_2_7_DB".KP[0].CMD.Reset THEN
	        "KP_2_7_DB".KP[0].CMD.Reset := FALSE;
	    END_IF;
	END_IF;
	
	    
END_FUNCTION

FUNCTION_BLOCK "KP_2_8"
{ S7_Optimized_Access := 'FALSE' }
VERSION : 0.1
   VAR 
      limit { S7_SetPoint := 'True'} : Int := 2;   // число задвижек в камере
      load : Int;   // отображаемые на экране настройки
      load_last : Int;
      KP : Array[0..10] of "DRV_AUMA";
      load_ok { S7_SetPoint := 'True'} : Bool;
   END_VAR

   VAR_TEMP 
      ID : Int;
      cnt : Int;
   END_VAR


BEGIN
	//дистанционный режим управления
	FOR #cnt := 1 TO #limit BY 1 DO
	    IF "Comm_SKV_3".To_SKV.Valves.Local[0] THEN
	        IF #KP[#cnt].CMD.Hand THEN
	            #KP[#cnt].CMD.Start_M := "Comm_SKV_3".From_SKV.Valves.REQ[#cnt];
	        END_IF;
	        IF "Comm_SKV_3".From_SKV.Valves.REQ[0] THEN
	            #KP[#cnt].CMD.Reset := TRUE;
	            #load := 10;
	        END_IF;
	    ELSE
	        "Comm_SKV_3".To_SKV.Valves.Local[#cnt] := #KP[#cnt].CMD.Start_M;
	    END_IF;
	END_FOR;
	
	//экранный буфер
	"Load_KP_2_8"(last := #load_last,
	              load := #load,
	              ok := #load_ok);
	IF "KP_Reset" THEN
	    #load := 10;
	END_IF;
	
	FOR #cnt := 1 TO #limit BY 1 DO
	    #ID := #KP[#cnt].CodeID;
	    #KP[#cnt].CMD.Local := NOT "AUMA_KP_2_8_DB".AUMA[#ID].Message.Sel_Dist;
	    #KP[#cnt].Alarm.Link := NOT "AUMA_KP_2_8_DB".AUMA[#ID].Link;
	    #KP[#cnt].Use.Enable := "AUMA_KP_2_8_DB".AUMA[#ID].Use;
	    #KP[#cnt].Name := "AUMA_KP_2_8_DB".AUMA[#ID].Name;
	    #KP[#cnt].Position := INT_TO_REAL("AUMA_KP_2_8_DB".AUMA[#ID].Position) / 10.0;
	    #KP[#cnt].FB.QF := "AUMA_KP_2_8_DB".AUMA[#ID].Message.NotReady;
	    #KP[#cnt].FB.KM_Open := "AUMA_KP_2_8_DB".AUMA[#ID].Message.Opening;
	    #KP[#cnt].FB.KM_Close := "AUMA_KP_2_8_DB".AUMA[#ID].Message.Closing;
	    #KP[#cnt].FB.Open := "AUMA_KP_2_8_DB".AUMA[#ID].Message.Open;
	    #KP[#cnt].FB.Close := "AUMA_KP_2_8_DB".AUMA[#ID].Message.Close;
	    #KP[#cnt]();
	    "AUMA_KP_2_8_DB".AUMA[#ID].Speed := #KP[#cnt].Speed;
	    "AUMA_KP_2_8_DB".AUMA[#ID].CMD.Open := #KP[#cnt].CMD_Open;
	    "AUMA_KP_2_8_DB".AUMA[#ID].CMD.Close := #KP[#cnt].CMD_Close;
	    IF "AUMA_KP_2_8_DB".AUMA[#ID].CMD.Open <> "AUMA_KP_2_8_DB".AUMA[#ID].CMD_last.Open THEN
	        "AUMA_KP_2_8_DB".AUMA[#ID].CMD_last.Open := "AUMA_KP_2_8_DB".AUMA[#ID].CMD.Open;
	        "AUMA_KP_2_8_DB".AUMA[#ID].Update := true;
	    END_IF;
	    IF "AUMA_KP_2_8_DB".AUMA[#ID].CMD.Close <> "AUMA_KP_2_8_DB".AUMA[#ID].CMD_last.Close THEN
	        "AUMA_KP_2_8_DB".AUMA[#ID].CMD_last.Close := "AUMA_KP_2_8_DB".AUMA[#ID].CMD.Close;
	        "AUMA_KP_2_8_DB".AUMA[#ID].Update := true;
	    END_IF;
	END_FOR;
END_FUNCTION_BLOCK

FUNCTION "Load_KP_2_8" : Void
{ S7_Optimized_Access := 'TRUE' }
VERSION : 0.1
   VAR_IN_OUT 
      ok : Bool;
      load : Int;
      last : Int;
   END_VAR


BEGIN
	//проверка загруженных данных
	IF #load <> #last THEN
	    #ok := FALSE;
	END_IF;
	
	//первичная загрузка данных
	IF NOT #ok THEN
	    "KP_2_8_DB".KP[0].CMD := "KP_2_8_DB".KP[#load].CMD;
	    "KP_2_8_DB".KP[0].Mode := "KP_2_8_DB".KP[#load].Mode;
	    "KP_2_8_DB".KP[0].Status := "KP_2_8_DB".KP[#load].Status;
	    "KP_2_8_DB".KP[0].FB := "KP_2_8_DB".KP[#load].FB;
	    "KP_2_8_DB".KP[0].Use := "KP_2_8_DB".KP[#load].Use;
	    "KP_2_8_DB".KP[0].Alarm := "KP_2_8_DB".KP[#load].Alarm;
	    "KP_2_8_DB".KP[0].Clock[0].SP := "KP_2_8_DB".KP[#load].Clock[0].SP;
	    "KP_2_8_DB".KP[0].Clock[0].Now := "KP_2_8_DB".KP[#load].Clock[0].Now;
	    "KP_2_8_DB".KP[0].Clock[1].SP := "KP_2_8_DB".KP[#load].Clock[1].SP;
	    "KP_2_8_DB".KP[0].Clock[1].Now := "KP_2_8_DB".KP[#load].Clock[1].Now;
	    "KP_2_8_DB".KP[0].Clock[2].SP := "KP_2_8_DB".KP[#load].Clock[2].SP;
	    "KP_2_8_DB".KP[0].Clock[2].Now := "KP_2_8_DB".KP[#load].Clock[2].Now;
	    "KP_2_8_DB".KP[0].Clock[3].SP := "KP_2_8_DB".KP[#load].Clock[3].SP;
	    "KP_2_8_DB".KP[0].Clock[3].Now := "KP_2_8_DB".KP[#load].Clock[3].Now;
	    "KP_2_8_DB".KP[0].Clock[4].SP := "KP_2_8_DB".KP[#load].Clock[4].SP;
	    "KP_2_8_DB".KP[0].Clock[4].Now := "KP_2_8_DB".KP[#load].Clock[4].Now;
	    "KP_2_8_DB".KP[0].CodeID := "KP_2_8_DB".KP[#load].CodeID;
	    "KP_2_8_DB".KP[0].Position := "KP_2_8_DB".KP[#load].Position;
	    "KP_2_8_DB".KP[0].Speed := "KP_2_8_DB".KP[#load].Speed;
	    "KP_2_8_DB".KP[0].Name := "KP_2_8_DB".KP[#load].Name;
	    #ok := true;
	    #last := #load;
	END_IF;
	
	//управление с панели
	IF #ok THEN
	    "KP_2_8_DB".KP[#load].CMD.Hand := "KP_2_8_DB".KP[0].CMD.Hand;
	    "KP_2_8_DB".KP[#load].CMD.Force := "KP_2_8_DB".KP[0].CMD.Force;
	    "KP_2_8_DB".KP[#load].CMD.Start_M := "KP_2_8_DB".KP[0].CMD.Start_M;
	    "KP_2_8_DB".KP[#load].CMD.Reset := "KP_2_8_DB".KP[0].CMD.Reset;
	    "KP_2_8_DB".KP[#load].Use := "KP_2_8_DB".KP[0].Use;
	    "KP_2_8_DB".KP[#load].Clock[0].SP := "KP_2_8_DB".KP[0].Clock[0].SP;
	    "KP_2_8_DB".KP[#load].Clock[1].SP := "KP_2_8_DB".KP[0].Clock[1].SP;
	    "KP_2_8_DB".KP[#load].Clock[2].SP := "KP_2_8_DB".KP[0].Clock[2].SP;
	    "KP_2_8_DB".KP[#load].Clock[3].SP := "KP_2_8_DB".KP[0].Clock[3].SP;
	    "KP_2_8_DB".KP[#load].Clock[4].SP := "KP_2_8_DB".KP[0].Clock[4].SP;
	    "KP_2_8_DB".KP[#load].CodeID := "KP_2_8_DB".KP[0].CodeID;
	    "KP_2_8_DB".KP[#load].Speed := "KP_2_8_DB".KP[0].Speed;
	    "KP_2_8_DB".KP[0].CMD.Local := "KP_2_8_DB".KP[#load].CMD.Local;
	    "KP_2_8_DB".KP[0].CMD.Lock := "KP_2_8_DB".KP[#load].CMD.Lock;
	    "KP_2_8_DB".KP[0].Mode := "KP_2_8_DB".KP[#load].Mode;
	    "KP_2_8_DB".KP[0].Status := "KP_2_8_DB".KP[#load].Status;
	    "KP_2_8_DB".KP[0].FB := "KP_2_8_DB".KP[#load].FB;
	    "KP_2_8_DB".KP[0].Alarm := "KP_2_8_DB".KP[#load].Alarm;
	    "KP_2_8_DB".KP[0].Clock[0].Now := "KP_2_8_DB".KP[#load].Clock[0].Now;
	    "KP_2_8_DB".KP[0].Clock[1].Now := "KP_2_8_DB".KP[#load].Clock[1].Now;
	    "KP_2_8_DB".KP[0].Clock[2].Now := "KP_2_8_DB".KP[#load].Clock[2].Now;
	    "KP_2_8_DB".KP[0].Clock[3].Now := "KP_2_8_DB".KP[#load].Clock[3].Now;
	    "KP_2_8_DB".KP[0].Clock[4].Now := "KP_2_8_DB".KP[#load].Clock[4].Now;
	    "KP_2_8_DB".KP[0].Position := "KP_2_8_DB".KP[#load].Position;
	    IF "KP_2_8_DB".KP[0].CMD.Reset THEN
	        "KP_2_8_DB".KP[0].CMD.Reset := FALSE;
	    END_IF;
	END_IF;
	
	    
END_FUNCTION

FUNCTION_BLOCK "KP_2_9"
{ S7_Optimized_Access := 'FALSE' }
VERSION : 0.1
   VAR 
      limit { S7_SetPoint := 'True'} : Int := 2;   // число задвижек в камере
      load : Int;   // отображаемые на экране настройки
      load_last : Int;
      KP : Array[0..10] of "DRV_AUMA";
      load_ok { S7_SetPoint := 'True'} : Bool;
   END_VAR

   VAR_TEMP 
      ID : Int;
      cnt : Int;
   END_VAR


BEGIN
	//дистанционный режим управления
	FOR #cnt := 1 TO #limit BY 1 DO
	    IF "Comm_SKV_12".To_SKV.Valves.Local[0] THEN
	        IF #KP[#cnt].CMD.Hand THEN
	            #KP[#cnt].CMD.Start_M := "Comm_SKV_12".From_SKV.Valves.REQ[#cnt];
	        END_IF;
	        IF "Comm_SKV_12".From_SKV.Valves.REQ[0] THEN
	            #KP[#cnt].CMD.Reset := TRUE;
	            #load := 10;
	        END_IF;
	    ELSE
	        "Comm_SKV_12".To_SKV.Valves.Local[#cnt] := #KP[#cnt].CMD.Start_M;
	    END_IF;
	END_FOR;
	
	//экранный буфер
	"Load_KP_2_9"(last := #load_last,
	              load := #load,
	              ok := #load_ok);
	IF "KP_Reset" THEN
	    #load := 10;
	END_IF;
	
	FOR #cnt := 1 TO #limit BY 1 DO
	    #ID := #KP[#cnt].CodeID;
	    #KP[#cnt].CMD.Local := NOT "AUMA_KP_2_9_DB".AUMA[#ID].Message.Sel_Dist;
	    #KP[#cnt].Alarm.Link := NOT "AUMA_KP_2_9_DB".AUMA[#ID].Link;
	    #KP[#cnt].Use.Enable := "AUMA_KP_2_9_DB".AUMA[#ID].Use;
	    #KP[#cnt].Name := "AUMA_KP_2_9_DB".AUMA[#ID].Name;
	    #KP[#cnt].Position := INT_TO_REAL("AUMA_KP_2_9_DB".AUMA[#ID].Position) / 10.0;
	    #KP[#cnt].FB.QF := "AUMA_KP_2_9_DB".AUMA[#ID].Message.NotReady;
	    #KP[#cnt].FB.KM_Open := "AUMA_KP_2_9_DB".AUMA[#ID].Message.Opening;
	    #KP[#cnt].FB.KM_Close := "AUMA_KP_2_9_DB".AUMA[#ID].Message.Closing;
	    #KP[#cnt].FB.Open := "AUMA_KP_2_9_DB".AUMA[#ID].Message.Open;
	    #KP[#cnt].FB.Close := "AUMA_KP_2_9_DB".AUMA[#ID].Message.Close;
	    #KP[#cnt]();
	    "AUMA_KP_2_9_DB".AUMA[#ID].Speed := #KP[#cnt].Speed;
	    "AUMA_KP_2_9_DB".AUMA[#ID].CMD.Open := #KP[#cnt].CMD_Open;
	    "AUMA_KP_2_9_DB".AUMA[#ID].CMD.Close := #KP[#cnt].CMD_Close;
	    IF "AUMA_KP_2_9_DB".AUMA[#ID].CMD.Open <> "AUMA_KP_2_9_DB".AUMA[#ID].CMD_last.Open THEN
	        "AUMA_KP_2_9_DB".AUMA[#ID].CMD_last.Open := "AUMA_KP_2_9_DB".AUMA[#ID].CMD.Open;
	        "AUMA_KP_2_9_DB".AUMA[#ID].Update := true;
	    END_IF;
	    IF "AUMA_KP_2_9_DB".AUMA[#ID].CMD.Close <> "AUMA_KP_2_9_DB".AUMA[#ID].CMD_last.Close THEN
	        "AUMA_KP_2_9_DB".AUMA[#ID].CMD_last.Close := "AUMA_KP_2_9_DB".AUMA[#ID].CMD.Close;
	        "AUMA_KP_2_9_DB".AUMA[#ID].Update := true;
	    END_IF;
	END_FOR;
END_FUNCTION_BLOCK

FUNCTION "Load_KP_2_9" : Void
{ S7_Optimized_Access := 'TRUE' }
VERSION : 0.1
   VAR_IN_OUT 
      ok : Bool;
      load : Int;
      last : Int;
   END_VAR


BEGIN
	//проверка загруженных данных
	IF #load <> #last THEN
	    #ok := FALSE;
	END_IF;
	
	//первичная загрузка данных
	IF NOT #ok THEN
	    "KP_2_9_DB".KP[0].CMD := "KP_2_9_DB".KP[#load].CMD;
	    "KP_2_9_DB".KP[0].Mode := "KP_2_9_DB".KP[#load].Mode;
	    "KP_2_9_DB".KP[0].Status := "KP_2_9_DB".KP[#load].Status;
	    "KP_2_9_DB".KP[0].FB := "KP_2_9_DB".KP[#load].FB;
	    "KP_2_9_DB".KP[0].Use := "KP_2_9_DB".KP[#load].Use;
	    "KP_2_9_DB".KP[0].Alarm := "KP_2_9_DB".KP[#load].Alarm;
	    "KP_2_9_DB".KP[0].Clock[0].SP := "KP_2_9_DB".KP[#load].Clock[0].SP;
	    "KP_2_9_DB".KP[0].Clock[0].Now := "KP_2_9_DB".KP[#load].Clock[0].Now;
	    "KP_2_9_DB".KP[0].Clock[1].SP := "KP_2_9_DB".KP[#load].Clock[1].SP;
	    "KP_2_9_DB".KP[0].Clock[1].Now := "KP_2_9_DB".KP[#load].Clock[1].Now;
	    "KP_2_9_DB".KP[0].Clock[2].SP := "KP_2_9_DB".KP[#load].Clock[2].SP;
	    "KP_2_9_DB".KP[0].Clock[2].Now := "KP_2_9_DB".KP[#load].Clock[2].Now;
	    "KP_2_9_DB".KP[0].Clock[3].SP := "KP_2_9_DB".KP[#load].Clock[3].SP;
	    "KP_2_9_DB".KP[0].Clock[3].Now := "KP_2_9_DB".KP[#load].Clock[3].Now;
	    "KP_2_9_DB".KP[0].Clock[4].SP := "KP_2_9_DB".KP[#load].Clock[4].SP;
	    "KP_2_9_DB".KP[0].Clock[4].Now := "KP_2_9_DB".KP[#load].Clock[4].Now;
	    "KP_2_9_DB".KP[0].CodeID := "KP_2_9_DB".KP[#load].CodeID;
	    "KP_2_9_DB".KP[0].Position := "KP_2_9_DB".KP[#load].Position;
	    "KP_2_9_DB".KP[0].Speed := "KP_2_9_DB".KP[#load].Speed;
	    "KP_2_9_DB".KP[0].Name := "KP_2_9_DB".KP[#load].Name;
	    #ok := true;
	    #last := #load;
	END_IF;
	
	//управление с панели
	IF #ok THEN
	    "KP_2_9_DB".KP[#load].CMD.Hand := "KP_2_9_DB".KP[0].CMD.Hand;
	    "KP_2_9_DB".KP[#load].CMD.Force := "KP_2_9_DB".KP[0].CMD.Force;
	    "KP_2_9_DB".KP[#load].CMD.Start_M := "KP_2_9_DB".KP[0].CMD.Start_M;
	    "KP_2_9_DB".KP[#load].CMD.Reset := "KP_2_9_DB".KP[0].CMD.Reset;
	    "KP_2_9_DB".KP[#load].Use := "KP_2_9_DB".KP[0].Use;
	    "KP_2_9_DB".KP[#load].Clock[0].SP := "KP_2_9_DB".KP[0].Clock[0].SP;
	    "KP_2_9_DB".KP[#load].Clock[1].SP := "KP_2_9_DB".KP[0].Clock[1].SP;
	    "KP_2_9_DB".KP[#load].Clock[2].SP := "KP_2_9_DB".KP[0].Clock[2].SP;
	    "KP_2_9_DB".KP[#load].Clock[3].SP := "KP_2_9_DB".KP[0].Clock[3].SP;
	    "KP_2_9_DB".KP[#load].Clock[4].SP := "KP_2_9_DB".KP[0].Clock[4].SP;
	    "KP_2_9_DB".KP[#load].CodeID := "KP_2_9_DB".KP[0].CodeID;
	    "KP_2_9_DB".KP[#load].Speed := "KP_2_9_DB".KP[0].Speed;
	    "KP_2_9_DB".KP[0].CMD.Local := "KP_2_9_DB".KP[#load].CMD.Local;
	    "KP_2_9_DB".KP[0].CMD.Lock := "KP_2_9_DB".KP[#load].CMD.Lock;
	    "KP_2_9_DB".KP[0].Mode := "KP_2_9_DB".KP[#load].Mode;
	    "KP_2_9_DB".KP[0].Status := "KP_2_9_DB".KP[#load].Status;
	    "KP_2_9_DB".KP[0].FB := "KP_2_9_DB".KP[#load].FB;
	    "KP_2_9_DB".KP[0].Alarm := "KP_2_9_DB".KP[#load].Alarm;
	    "KP_2_9_DB".KP[0].Clock[0].Now := "KP_2_9_DB".KP[#load].Clock[0].Now;
	    "KP_2_9_DB".KP[0].Clock[1].Now := "KP_2_9_DB".KP[#load].Clock[1].Now;
	    "KP_2_9_DB".KP[0].Clock[2].Now := "KP_2_9_DB".KP[#load].Clock[2].Now;
	    "KP_2_9_DB".KP[0].Clock[3].Now := "KP_2_9_DB".KP[#load].Clock[3].Now;
	    "KP_2_9_DB".KP[0].Clock[4].Now := "KP_2_9_DB".KP[#load].Clock[4].Now;
	    "KP_2_9_DB".KP[0].Position := "KP_2_9_DB".KP[#load].Position;
	    IF "KP_2_9_DB".KP[0].CMD.Reset THEN
	        "KP_2_9_DB".KP[0].CMD.Reset := FALSE;
	    END_IF;
	END_IF;
	
	    
END_FUNCTION

FUNCTION_BLOCK "KP_2_10"
{ S7_Optimized_Access := 'FALSE' }
VERSION : 0.1
   VAR 
      limit { S7_SetPoint := 'True'} : Int := 2;   // число задвижек в камере
      load : Int;   // отображаемые на экране настройки
      load_last : Int;
      KP : Array[0..10] of "DRV_AUMA";
      load_ok { S7_SetPoint := 'True'} : Bool;
   END_VAR

   VAR_TEMP 
      ID : Int;
      cnt : Int;
   END_VAR


BEGIN
	//дистанционный режим управления
	FOR #cnt := 1 TO #limit BY 1 DO
	    IF "Comm_SKV_15".To_SKV.Valves.Local[0] THEN
	        IF #KP[#cnt].CMD.Hand THEN
	            #KP[#cnt].CMD.Start_M := "Comm_SKV_15".From_SKV.Valves.REQ[#cnt];
	        END_IF;
	        IF "Comm_SKV_15".From_SKV.Valves.REQ[0] THEN
	            #KP[#cnt].CMD.Reset := TRUE;
	            #load := 10;
	        END_IF;
	    ELSE
	        "Comm_SKV_15".To_SKV.Valves.Local[#cnt] := #KP[#cnt].CMD.Start_M;
	    END_IF;
	END_FOR;
	
	//экранный буфер
	"Load_KP_2_10"(last := #load_last,
	              load := #load,
	              ok := #load_ok);
	IF "KP_Reset" THEN
	    #load := 10;
	END_IF;
	
	FOR #cnt := 1 TO #limit BY 1 DO
	    #ID := #KP[#cnt].CodeID;
	    #KP[#cnt].CMD.Local := NOT "AUMA_KP_2_10_DB".AUMA[#ID].Message.Sel_Dist;
	    #KP[#cnt].Alarm.Link := NOT "AUMA_KP_2_10_DB".AUMA[#ID].Link;
	    #KP[#cnt].Use.Enable := "AUMA_KP_2_10_DB".AUMA[#ID].Use;
	    #KP[#cnt].Name := "AUMA_KP_2_10_DB".AUMA[#ID].Name;
	    #KP[#cnt].Position := INT_TO_REAL("AUMA_KP_2_10_DB".AUMA[#ID].Position) / 10.0;
	    #KP[#cnt].FB.QF := "AUMA_KP_2_10_DB".AUMA[#ID].Message.NotReady;
	    #KP[#cnt].FB.KM_Open := "AUMA_KP_2_10_DB".AUMA[#ID].Message.Opening;
	    #KP[#cnt].FB.KM_Close := "AUMA_KP_2_10_DB".AUMA[#ID].Message.Closing;
	    #KP[#cnt].FB.Open := "AUMA_KP_2_10_DB".AUMA[#ID].Message.Open;
	    #KP[#cnt].FB.Close := "AUMA_KP_2_10_DB".AUMA[#ID].Message.Close;
	    #KP[#cnt]();
	    "AUMA_KP_2_10_DB".AUMA[#ID].Speed := #KP[#cnt].Speed;
	    "AUMA_KP_2_10_DB".AUMA[#ID].CMD.Open := #KP[#cnt].CMD_Open;
	    "AUMA_KP_2_10_DB".AUMA[#ID].CMD.Close := #KP[#cnt].CMD_Close;
	    IF "AUMA_KP_2_10_DB".AUMA[#ID].CMD.Open <> "AUMA_KP_2_10_DB".AUMA[#ID].CMD_last.Open THEN
	        "AUMA_KP_2_10_DB".AUMA[#ID].CMD_last.Open := "AUMA_KP_2_10_DB".AUMA[#ID].CMD.Open;
	        "AUMA_KP_2_10_DB".AUMA[#ID].Update := true;
	    END_IF;
	    IF "AUMA_KP_2_10_DB".AUMA[#ID].CMD.Close <> "AUMA_KP_2_10_DB".AUMA[#ID].CMD_last.Close THEN
	        "AUMA_KP_2_10_DB".AUMA[#ID].CMD_last.Close := "AUMA_KP_2_10_DB".AUMA[#ID].CMD.Close;
	        "AUMA_KP_2_10_DB".AUMA[#ID].Update := true;
	    END_IF;
	END_FOR;
END_FUNCTION_BLOCK

FUNCTION "Load_KP_2_10" : Void
{ S7_Optimized_Access := 'TRUE' }
VERSION : 0.1
   VAR_IN_OUT 
      ok : Bool;
      load : Int;
      last : Int;
   END_VAR


